SPLINE
SPL {X  -138.661, Y  +302.689, Z    +0.000, E1  +316.811, E3 -159767.577}
SPL {X  -154.202, Y  +339.857, Z    +0.000, E1  +330.366, E3 -159785.230}
SPL {X  -158.556, Y  +361.128, Z    +0.000, E1  +342.470, E3 -159789.751}
SPL {X  -159.866, Y  +376.206, Z    +0.000, E1  +353.031, E3 -159791.280}
SPL {X  -159.990, Y  +384.326, Z    +0.000, E1  +359.760, E3 -159791.553}
SPL {X  -159.990, Y  +385.649, Z    +0.000, E1  +361.559, E3 -159791.566}
SPL {X  -159.990, Y  +388.306, Z    +0.000, E1  +365.901, E3 -159791.637}
SPL {X  -159.990, Y  +392.624, Z    +0.000, E1  +373.655, E3 -159791.887}
SPL {X  -159.990, Y  +398.511, Z    +0.000, E1  +384.979, E3 -159792.467}
SPL {X  -159.990, Y  +405.629, Z    +0.000, E1  +396.596, E3 -159793.598}
SPL {X  -159.990, Y  +418.631, Z    +0.000, E1  +410.627, E3 -159796.545}
SPL {X  -159.990, Y  +468.459, Z    +0.000, E1  +425.348, E3 -159816.088}
SPL {X  -159.990, Y  +601.948, Z    +0.000, E1  +428.261, E3 -159902.214}
SPL {X  -159.990, Y  +614.867, Z    +0.000, E1  +428.239, E3 -159913.213}
SPL {X  -159.990, Y  +627.954, Z    +0.000, E1  +428.256, E3 -159924.257}
SPL {X  -159.990, Y  +640.176, Z    +0.000, E1  +428.239, E3 -159934.636}
SPL {X  -159.990, Y  +653.116, Z    +0.000, E1  +428.255, E3 -159945.568}
SPL {X  -159.990, Y  +665.424, Z    +0.000, E1  +428.236, E3 -159956.032}
SPL {X  -159.958, Y  +674.683, Z    +0.000, E1  +428.238, E3 -159963.881}
SPL {X  -159.269, Y  +686.675, Z    +0.000, E1  +428.163, E3 -159974.758}
SPL {X  -158.119, Y  +695.895, Z    +0.000, E1  +428.003, E3 -159983.799}
SPL {X  -156.550, Y  +704.498, Z    +0.000, E1  +427.821, E3 -159992.689}
SPL {X  -153.468, Y  +716.715, Z    +0.000, E1  +427.444, E3 -160006.152}
SPL {X  -149.840, Y  +727.578, Z    +0.000, E1  +426.935, E3 -160019.028}
SPL {X  -145.768, Y  +737.444, Z    +0.000, E1  +426.379, E3 -160031.330}
SPL {X  -141.751, Y  +745.686, Z    +0.000, E1  +425.756, E3 -160042.146}
SPL {X  -138.928, Y  +750.847, Z    +0.000, E1  +425.305, E3 -160049.116}
SPL {X  -136.328, Y  +755.234, Z    +0.000, E1  +424.898, E3 -160055.106}
SPL {X  -132.717, Y  +760.848, Z    +0.000, E1  +424.322, E3 -160062.879}
SPL {X  -128.512, Y  +766.796, Z    +0.000, E1  +423.597, E3 -160071.234}
SPL {X   -99.023, Y  +797.163, Z    +0.000, E1  +413.965, E3 -160173.063}
ENDSPLINE

SPLINE
SPL {X  -130.021, Y  +764.727, Z    +0.000, E1  +405.990, E3 -160312.582}
SPL {X  -148.409, Y  +731.264, Z    +0.000, E1  +396.685, E3 -160336.296}
SPL {X  -155.017, Y  +711.078, Z    +0.000, E1  +387.846, E3 -160343.357}
SPL {X  -158.217, Y  +695.254, Z    +0.000, E1  +378.896, E3 -160346.800}
SPL {X  -159.762, Y  +680.037, Z    +0.000, E1  +368.585, E3 -160348.517}
SPL {X  -159.990, Y  +669.745, Z    +0.000, E1  +360.389, E3 -160348.939}
SPL {X  -159.990, Y  +666.879, Z    +0.000, E1  +356.292, E3 -160348.990}
SPL {X  -159.990, Y  +662.620, Z    +0.000, E1  +348.758, E3 -160349.191}
SPL {X  -159.990, Y  +657.714, Z    +0.000, E1  +339.502, E3 -160349.612}
SPL {X  -159.990, Y  +651.038, Z    +0.000, E1  +327.797, E3 -160350.515}
SPL {X  -159.990, Y  +637.243, Z    +0.000, E1  +311.500, E3 -160353.640}
SPL {X  -159.990, Y  +579.875, Z    +0.000, E1  +294.421, E3 -160376.499}
SPL {X  -159.990, Y  +453.091, Z    +0.000, E1  +291.862, E3 -160459.468}
SPL {X  -159.990, Y  +439.299, Z    +0.000, E1  +291.885, E3 -160471.281}
SPL {X  -159.990, Y  +424.060, Z    +0.000, E1  +291.860, E3 -160484.229}
SPL {X  -159.990, Y  +408.047, Z    +0.000, E1  +291.885, E3 -160497.935}
SPL {X  -159.990, Y  +395.904, Z    +0.000, E1  +291.881, E3 -160508.271}
SPL {X  -157.896, Y  +356.699, Z    +0.000, E1  +289.725, E3 -160520.581}
SPL {X  -156.475, Y  +349.148, Z    +0.000, E1  +290.612, E3 -160534.045}
SPL {X  -155.960, Y  +346.816, Z    +0.000, E1  +291.495, E3 -160543.206}
SPL {X  -154.913, Y  +342.515, Z    +0.000, E1  +292.501, E3 -160555.220}
SPL {X  -152.032, Y  +332.668, Z    +0.000, E1  +292.988, E3 -160567.211}
SPL {X  -149.782, Y  +326.266, Z    +0.000, E1  +293.308, E3 -160574.951}
SPL {X  -147.566, Y  +320.686, Z    +0.000, E1  +293.613, E3 -160581.888}
SPL {X  -144.472, Y  +313.764, Z    +0.000, E1  +294.050, E3 -160590.757}
SPL {X  -140.755, Y  +306.442, Z    +0.000, E1  +294.606, E3 -160600.472}
SPL {X  -137.162, Y  +300.138, Z    +0.000, E1  +295.180, E3 -160609.080}
SPL {X  -132.996, Y  +293.568, Z    +0.000, E1  +295.842, E3 -160618.215}
SPL {X  -128.628, Y  +287.360, Z    +0.000, E1  +296.617, E3 -160627.016}
SPL {X   -99.903, Y  +257.535, Z    +0.000, E1  +308.539, E3 -160775.879}
ENDSPLINE

SPLINE
SPL {X  -141.433, Y  +307.709, Z    +0.000, E1  +318.157, E3 -160885.676}
SPL {X  -154.202, Y  +339.857, Z    +0.000, E1  +330.366, E3 -160899.515}
SPL {X  -158.556, Y  +361.128, Z    +0.000, E1  +342.470, E3 -160904.037}
SPL {X  -159.663, Y  +372.278, Z    +0.000, E1  +350.186, E3 -160905.319}
SPL {X  -159.986, Y  +381.388, Z    +0.000, E1  +357.201, E3 -160905.790}
SPL {X  -159.990, Y  +384.492, Z    +0.000, E1  +359.986, E3 -160905.840}
SPL {X  -159.990, Y  +385.649, Z    +0.000, E1  +361.559, E3 -160905.851}
SPL {X  -159.990, Y  +389.563, Z    +0.000, E1  +367.931, E3 -160905.984}
SPL {X  -159.990, Y  +396.421, Z    +0.000, E1  +380.831, E3 -160906.529}
SPL {X  -159.990, Y  +405.629, Z    +0.000, E1  +396.596, E3 -160907.883}
SPL {X  -159.990, Y  +418.631, Z    +0.000, E1  +410.627, E3 -160910.831}
SPL {X  -159.990, Y  +468.459, Z    +0.000, E1  +425.348, E3 -160930.374}
SPL {X  -159.990, Y  +601.948, Z    +0.000, E1  +428.261, E3 -161016.500}
SPL {X  -159.990, Y  +619.726, Z    +0.000, E1  +428.262, E3 -161031.561}
SPL {X  -159.990, Y  +636.530, Z    +0.000, E1  +428.257, E3 -161045.797}
SPL {X  -159.990, Y  +648.825, Z    +0.000, E1  +428.237, E3 -161056.256}
SPL {X  -159.990, Y  +661.441, Z    +0.000, E1  +428.256, E3 -161066.904}
SPL {X  -159.958, Y  +674.683, Z    +0.000, E1  +428.238, E3 -161078.166}
SPL {X  -159.269, Y  +686.675, Z    +0.000, E1  +428.163, E3 -161089.044}
SPL {X  -157.606, Y  +699.018, Z    +0.000, E1  +427.957, E3 -161101.228}
SPL {X  -155.210, Y  +710.317, Z    +0.000, E1  +427.656, E3 -161113.268}
SPL {X  -152.048, Y  +721.282, Z    +0.000, E1  +427.243, E3 -161125.760}
SPL {X  -148.485, Y  +731.073, Z    +0.000, E1  +426.748, E3 -161137.609}
SPL {X  -145.075, Y  +738.953, Z    +0.000, E1  +426.252, E3 -161147.601}
SPL {X  -141.751, Y  +745.686, Z    +0.000, E1  +425.756, E3 -161156.432}
SPL {X  -138.928, Y  +750.847, Z    +0.000, E1  +425.305, E3 -161163.401}
SPL {X  -136.328, Y  +755.234, Z    +0.000, E1  +424.898, E3 -161169.392}
SPL {X  -132.717, Y  +760.848, Z    +0.000, E1  +424.322, E3 -161177.165}
SPL {X  -128.512, Y  +766.796, Z    +0.000, E1  +423.597, E3 -161185.519}
SPL {X   -99.023, Y  +797.163, Z    +0.000, E1  +413.965, E3 -161287.349}
ENDSPLINE

SPLINE
SPL {X  -130.021, Y  +764.727, Z    +0.000, E1  +405.990, E3 -161426.868}
SPL {X  -148.409, Y  +731.264, Z    +0.000, E1  +396.685, E3 -161450.582}
SPL {X  -155.017, Y  +711.078, Z    +0.000, E1  +387.846, E3 -161457.643}
SPL {X  -158.217, Y  +695.254, Z    +0.000, E1  +378.896, E3 -161461.086}
SPL {X  -159.762, Y  +680.037, Z    +0.000, E1  +368.585, E3 -161462.802}
SPL {X  -159.990, Y  +671.255, Z    +0.000, E1  +361.602, E3 -161463.208}
SPL {X  -159.990, Y  +669.426, Z    +0.000, E1  +359.932, E3 -161463.228}
SPL {X  -159.990, Y  +666.879, Z    +0.000, E1  +356.292, E3 -161463.276}
SPL {X  -159.990, Y  +662.620, Z    +0.000, E1  +348.758, E3 -161463.477}
SPL {X  -159.990, Y  +657.714, Z    +0.000, E1  +339.502, E3 -161463.898}
SPL {X  -159.990, Y  +651.038, Z    +0.000, E1  +327.797, E3 -161464.800}
SPL {X  -159.990, Y  +637.243, Z    +0.000, E1  +311.500, E3 -161467.926}
SPL {X  -159.990, Y  +579.875, Z    +0.000, E1  +294.421, E3 -161490.784}
SPL {X  -159.990, Y  +458.824, Z    +0.000, E1  +291.885, E3 -161568.920}
SPL {X  -159.990, Y  +443.948, Z    +0.000, E1  +291.858, E3 -161581.543}
SPL {X  -159.990, Y  +424.060, Z    +0.000, E1  +291.860, E3 -161598.515}
SPL {X  -159.990, Y  +408.047, Z    +0.000, E1  +291.885, E3 -161612.221}
SPL {X  -159.990, Y  +395.904, Z    +0.000, E1  +291.881, E3 -161622.557}
SPL {X  -157.896, Y  +356.699, Z    +0.000, E1  +289.725, E3 -161634.866}
SPL {X  -156.475, Y  +349.148, Z    +0.000, E1  +290.612, E3 -161648.330}
SPL {X  -155.786, Y  +346.063, Z    +0.000, E1  +291.892, E3 -161661.625}
SPL {X  -154.401, Y  +340.583, Z    +0.000, E1  +292.675, E3 -161672.322}
SPL {X  -152.032, Y  +332.668, Z    +0.000, E1  +292.988, E3 -161681.497}
SPL {X  -148.460, Y  +322.864, Z    +0.000, E1  +293.452, E3 -161693.380}
SPL {X  -144.472, Y  +313.764, Z    +0.000, E1  +294.050, E3 -161705.043}
SPL {X  -140.755, Y  +306.442, Z    +0.000, E1  +294.606, E3 -161714.758}
SPL {X  -137.162, Y  +300.138, Z    +0.000, E1  +295.180, E3 -161723.366}
SPL {X  -132.996, Y  +293.568, Z    +0.000, E1  +295.842, E3 -161732.500}
SPL {X  -128.628, Y  +287.360, Z    +0.000, E1  +296.617, E3 -161741.301}
SPL {X   -98.696, Y  +256.580, Z    +0.000, E1  +308.006, E3 -161878.420}
ENDSPLINE

SPLINE
SPL {X  -138.661, Y  +302.689, Z    +0.000, E1  +316.811, E3 -161996.148}
SPL {X  -154.202, Y  +339.857, Z    +0.000, E1  +330.366, E3 -162013.801}
SPL {X  -158.556, Y  +361.128, Z    +0.000, E1  +342.470, E3 -162018.323}
SPL {X  -159.866, Y  +376.206, Z    +0.000, E1  +353.031, E3 -162019.852}
SPL {X  -159.990, Y  +384.789, Z    +0.000, E1  +360.146, E3 -162020.129}
SPL {X  -159.990, Y  +389.563, Z    +0.000, E1  +367.931, E3 -162020.269}
SPL {X  -159.990, Y  +396.421, Z    +0.000, E1  +380.831, E3 -162020.814}
SPL {X  -159.990, Y  +405.629, Z    +0.000, E1  +396.596, E3 -162022.169}
SPL {X  -159.990, Y  +417.919, Z    +0.000, E1  +410.108, E3 -162024.895}
SPL {X  -159.990, Y  +464.219, Z    +0.000, E1  +424.792, E3 -162042.954}
SPL {X  -159.990, Y  +601.948, Z    +0.000, E1  +428.261, E3 -162130.786}
SPL {X  -159.990, Y  +614.867, Z    +0.000, E1  +428.239, E3 -162141.784}
SPL {X  -159.990, Y  +627.954, Z    +0.000, E1  +428.256, E3 -162152.829}
SPL {X  -159.990, Y  +640.176, Z    +0.000, E1  +428.239, E3 -162163.207}
SPL {X  -159.990, Y  +653.116, Z    +0.000, E1  +428.255, E3 -162174.139}
SPL {X  -159.990, Y  +665.424, Z    +0.000, E1  +428.236, E3 -162184.603}
SPL {X  -159.958, Y  +674.683, Z    +0.000, E1  +428.238, E3 -162192.452}
SPL {X  -159.269, Y  +686.675, Z    +0.000, E1  +428.163, E3 -162203.330}
SPL {X  -157.606, Y  +699.018, Z    +0.000, E1  +427.957, E3 -162215.513}
SPL {X  -155.210, Y  +710.317, Z    +0.000, E1  +427.656, E3 -162227.553}
SPL {X  -152.048, Y  +721.282, Z    +0.000, E1  +427.243, E3 -162240.046}
SPL {X  -148.485, Y  +731.073, Z    +0.000, E1  +426.748, E3 -162251.895}
SPL {X  -145.075, Y  +738.953, Z    +0.000, E1  +426.252, E3 -162261.887}
SPL {X  -141.751, Y  +745.686, Z    +0.000, E1  +425.756, E3 -162270.718}
SPL {X  -138.928, Y  +750.847, Z    +0.000, E1  +425.305, E3 -162277.687}
SPL {X  -136.328, Y  +755.234, Z    +0.000, E1  +424.898, E3 -162283.677}
SPL {X  -132.717, Y  +760.848, Z    +0.000, E1  +424.322, E3 -162291.450}
SPL {X  -128.512, Y  +766.796, Z    +0.000, E1  +423.597, E3 -162299.805}
SPL {X   -99.023, Y  +797.163, Z    +0.000, E1  +413.965, E3 -162401.635}
ENDSPLINE

SPLINE
SPL {X  -130.021, Y  +764.727, Z    +0.000, E1  +405.990, E3 -162541.154}
SPL {X  -148.409, Y  +731.264, Z    +0.000, E1  +396.685, E3 -162564.867}
SPL {X  -155.017, Y  +711.078, Z    +0.000, E1  +387.846, E3 -162571.928}
SPL {X  -158.217, Y  +695.254, Z    +0.000, E1  +378.896, E3 -162575.371}
SPL {X  -159.762, Y  +680.037, Z    +0.000, E1  +368.585, E3 -162577.088}
SPL {X  -159.990, Y  +671.255, Z    +0.000, E1  +361.602, E3 -162577.494}
SPL {X  -159.990, Y  +669.148, Z    +0.000, E1  +359.679, E3 -162577.516}
SPL {X  -159.990, Y  +666.130, Z    +0.000, E1  +354.946, E3 -162577.582}
SPL {X  -159.990, Y  +662.620, Z    +0.000, E1  +348.758, E3 -162577.762}
SPL {X  -159.990, Y  +657.714, Z    +0.000, E1  +339.502, E3 -162578.184}
SPL {X  -159.990, Y  +651.038, Z    +0.000, E1  +327.797, E3 -162579.086}
SPL {X  -159.990, Y  +637.243, Z    +0.000, E1  +311.500, E3 -162582.211}
SPL {X  -159.990, Y  +579.875, Z    +0.000, E1  +294.421, E3 -162605.070}
SPL {X  -159.990, Y  +453.091, Z    +0.000, E1  +291.862, E3 -162688.039}
SPL {X  -159.990, Y  +439.299, Z    +0.000, E1  +291.885, E3 -162699.852}
SPL {X  -159.990, Y  +424.060, Z    +0.000, E1  +291.860, E3 -162712.800}
SPL {X  -159.990, Y  +408.047, Z    +0.000, E1  +291.885, E3 -162726.507}
SPL {X  -159.990, Y  +395.904, Z    +0.000, E1  +291.881, E3 -162736.843}
SPL {X  -157.896, Y  +356.699, Z    +0.000, E1  +289.725, E3 -162749.152}
SPL {X  -156.475, Y  +349.148, Z    +0.000, E1  +290.612, E3 -162762.616}
SPL {X  -155.786, Y  +346.063, Z    +0.000, E1  +291.892, E3 -162775.911}
SPL {X  -154.401, Y  +340.583, Z    +0.000, E1  +292.675, E3 -162786.607}
SPL {X  -152.032, Y  +332.668, Z    +0.000, E1  +292.988, E3 -162795.783}
SPL {X  -149.782, Y  +326.266, Z    +0.000, E1  +293.308, E3 -162803.523}
SPL {X  -146.798, Y  +318.884, Z    +0.000, E1  +293.699, E3 -162812.703}
SPL {X  -143.755, Y  +312.276, Z    +0.000, E1  +294.175, E3 -162821.313}
SPL {X  -140.755, Y  +306.442, Z    +0.000, E1  +294.606, E3 -162829.044}
SPL {X  -137.162, Y  +300.138, Z    +0.000, E1  +295.180, E3 -162837.652}
SPL {X  -134.303, Y  +295.555, Z    +0.000, E1  +295.659, E3 -162844.033}
SPL {X  -132.067, Y  +292.194, Z    +0.000, E1  +296.034, E3 -162848.764}
SPL {X  -128.628, Y  +287.360, Z    +0.000, E1  +296.617, E3 -162855.587}
SPL {X   -99.903, Y  +257.535, Z    +0.000, E1  +308.539, E3 -163004.450}
ENDSPLINE

SPLINE
SPL {X  -141.433, Y  +307.709, Z    +0.000, E1  +318.157, E3 -163114.247}
SPL {X  -151.246, Y  +330.333, Z    +0.000, E1  +326.099, E3 -163125.138}
SPL {X  -155.793, Y  +346.095, Z    +0.000, E1  +333.603, E3 -163129.796}
SPL {X  -158.556, Y  +361.128, Z    +0.000, E1  +342.470, E3 -163132.609}
SPL {X  -159.866, Y  +376.206, Z    +0.000, E1  +353.031, E3 -163134.138}
SPL {X  -159.990, Y  +384.326, Z    +0.000, E1  +359.760, E3 -163134.410}
SPL {X  -159.990, Y  +385.649, Z    +0.000, E1  +361.559, E3 -163134.423}
SPL {X  -159.990, Y  +388.306, Z    +0.000, E1  +365.901, E3 -163134.494}
SPL {X  -159.990, Y  +392.624, Z    +0.000, E1  +373.655, E3 -163134.744}
SPL {X  -159.990, Y  +398.511, Z    +0.000, E1  +384.979, E3 -163135.324}
SPL {X  -159.990, Y  +405.629, Z    +0.000, E1  +396.596, E3 -163136.455}
SPL {X  -159.990, Y  +418.631, Z    +0.000, E1  +410.627, E3 -163139.402}
SPL {X  -159.990, Y  +468.459, Z    +0.000, E1  +425.348, E3 -163158.945}
SPL {X  -159.990, Y  +601.948, Z    +0.000, E1  +428.261, E3 -163245.071}
SPL {X  -159.990, Y  +619.726, Z    +0.000, E1  +428.262, E3 -163260.132}
SPL {X  -159.990, Y  +636.530, Z    +0.000, E1  +428.257, E3 -163274.368}
SPL {X  -159.990, Y  +648.825, Z    +0.000, E1  +428.237, E3 -163284.827}
SPL {X  -159.990, Y  +661.441, Z    +0.000, E1  +428.256, E3 -163295.475}
SPL {X  -159.958, Y  +674.683, Z    +0.000, E1  +428.238, E3 -163306.738}
SPL {X  -159.269, Y  +686.675, Z    +0.000, E1  +428.163, E3 -163317.615}
SPL {X  -157.606, Y  +699.018, Z    +0.000, E1  +427.957, E3 -163329.799}
SPL {X  -155.210, Y  +710.317, Z    +0.000, E1  +427.656, E3 -163341.839}
SPL {X  -152.048, Y  +721.282, Z    +0.000, E1  +427.243, E3 -163354.332}
SPL {X  -148.485, Y  +731.073, Z    +0.000, E1  +426.748, E3 -163366.181}
SPL {X  -145.075, Y  +738.953, Z    +0.000, E1  +426.252, E3 -163376.172}
SPL {X  -141.751, Y  +745.686, Z    +0.000, E1  +425.756, E3 -163385.003}
SPL {X  -138.928, Y  +750.847, Z    +0.000, E1  +425.305, E3 -163391.973}
SPL {X  -136.328, Y  +755.234, Z    +0.000, E1  +424.898, E3 -163397.963}
SPL {X  -132.717, Y  +760.848, Z    +0.000, E1  +424.322, E3 -163405.736}
SPL {X  -128.512, Y  +766.796, Z    +0.000, E1  +423.597, E3 -163414.091}
SPL {X   -99.023, Y  +797.163, Z    +0.000, E1  +413.965, E3 -163515.920}
ENDSPLINE

SPLINE
SPL {X  -130.021, Y  +764.727, Z    +0.000, E1  +405.990, E3 -163655.440}
SPL {X  -148.409, Y  +731.264, Z    +0.000, E1  +396.685, E3 -163679.153}
SPL {X  -155.017, Y  +711.078, Z    +0.000, E1  +387.846, E3 -163686.214}
SPL {X  -158.217, Y  +695.254, Z    +0.000, E1  +378.896, E3 -163689.657}
SPL {X  -159.762, Y  +680.037, Z    +0.000, E1  +368.585, E3 -163691.374}
SPL {X  -159.990, Y  +671.255, Z    +0.000, E1  +361.602, E3 -163691.779}
SPL {X  -159.990, Y  +669.426, Z    +0.000, E1  +359.932, E3 -163691.799}
SPL {X  -159.990, Y  +666.879, Z    +0.000, E1  +356.292, E3 -163691.847}
SPL {X  -159.990, Y  +662.620, Z    +0.000, E1  +348.758, E3 -163692.048}
SPL {X  -159.990, Y  +657.714, Z    +0.000, E1  +339.502, E3 -163692.469}
SPL {X  -159.990, Y  +651.038, Z    +0.000, E1  +327.797, E3 -163693.372}
SPL {X  -159.990, Y  +637.243, Z    +0.000, E1  +311.500, E3 -163696.497}
SPL {X  -159.990, Y  +579.875, Z    +0.000, E1  +294.421, E3 -163719.356}
SPL {X  -159.990, Y  +453.091, Z    +0.000, E1  +291.862, E3 -163802.325}
SPL {X  -159.990, Y  +434.933, Z    +0.000, E1  +291.864, E3 -163817.819}
SPL {X  -159.990, Y  +420.071, Z    +0.000, E1  +291.886, E3 -163830.545}
SPL {X  -159.990, Y  +408.047, Z    +0.000, E1  +291.885, E3 -163840.792}
SPL {X  -159.990, Y  +395.904, Z    +0.000, E1  +291.881, E3 -163851.128}
SPL {X  -157.896, Y  +356.699, Z    +0.000, E1  +289.725, E3 -163863.438}
SPL {X  -156.475, Y  +349.148, Z    +0.000, E1  +290.612, E3 -163876.902}
SPL {X  -155.786, Y  +346.063, Z    +0.000, E1  +291.892, E3 -163890.196}
SPL {X  -153.671, Y  +337.981, Z    +0.000, E1  +292.746, E3 -163903.816}
SPL {X  -150.407, Y  +327.960, Z    +0.000, E1  +293.203, E3 -163915.705}
SPL {X  -146.798, Y  +318.884, Z    +0.000, E1  +293.699, E3 -163926.989}
SPL {X  -142.741, Y  +310.238, Z    +0.000, E1  +294.301, E3 -163938.248}
SPL {X  -139.838, Y  +304.768, Z    +0.000, E1  +294.773, E3 -163945.631}
SPL {X  -137.162, Y  +300.138, Z    +0.000, E1  +295.180, E3 -163951.937}
SPL {X  -132.996, Y  +293.568, Z    +0.000, E1  +295.842, E3 -163961.072}
SPL {X  -128.628, Y  +287.360, Z    +0.000, E1  +296.617, E3 -163969.873}
SPL {X   -98.696, Y  +256.580, Z    +0.000, E1  +308.006, E3 -164106.991}
ENDSPLINE

SPLINE
SPL {X  -138.661, Y  +302.689, Z    +0.000, E1  +316.811, E3 -164224.720}
SPL {X  -154.202, Y  +339.857, Z    +0.000, E1  +330.366, E3 -164242.373}
SPL {X  -158.556, Y  +361.128, Z    +0.000, E1  +342.470, E3 -164246.894}
SPL {X  -159.663, Y  +372.278, Z    +0.000, E1  +350.186, E3 -164248.176}
SPL {X  -159.986, Y  +381.388, Z    +0.000, E1  +357.201, E3 -164248.647}
SPL {X  -159.990, Y  +384.492, Z    +0.000, E1  +359.986, E3 -164248.697}
SPL {X  -159.990, Y  +385.649, Z    +0.000, E1  +361.559, E3 -164248.709}
SPL {X  -159.990, Y  +389.563, Z    +0.000, E1  +367.931, E3 -164248.841}
SPL {X  -159.990, Y  +396.421, Z    +0.000, E1  +380.831, E3 -164249.386}
SPL {X  -159.990, Y  +405.629, Z    +0.000, E1  +396.596, E3 -164250.740}
SPL {X  -159.990, Y  +418.631, Z    +0.000, E1  +410.627, E3 -164253.688}
SPL {X  -159.990, Y  +468.459, Z    +0.000, E1  +425.348, E3 -164273.231}
SPL {X  -159.990, Y  +601.948, Z    +0.000, E1  +428.261, E3 -164359.357}
SPL {X  -159.990, Y  +619.726, Z    +0.000, E1  +428.262, E3 -164374.418}
SPL {X  -159.990, Y  +636.530, Z    +0.000, E1  +428.257, E3 -164388.654}
SPL {X  -159.990, Y  +648.825, Z    +0.000, E1  +428.237, E3 -164399.113}
SPL {X  -159.990, Y  +661.441, Z    +0.000, E1  +428.256, E3 -164409.761}
SPL {X  -159.958, Y  +674.683, Z    +0.000, E1  +428.238, E3 -164421.024}
SPL {X  -159.269, Y  +686.675, Z    +0.000, E1  +428.163, E3 -164431.901}
SPL {X  -158.119, Y  +695.895, Z    +0.000, E1  +428.003, E3 -164440.942}
SPL {X  -156.550, Y  +704.498, Z    +0.000, E1  +427.821, E3 -164449.832}
SPL {X  -154.561, Y  +712.826, Z    +0.000, E1  +427.549, E3 -164458.963}
SPL {X  -152.048, Y  +721.282, Z    +0.000, E1  +427.243, E3 -164468.617}
SPL {X  -148.485, Y  +731.073, Z    +0.000, E1  +426.748, E3 -164480.466}
SPL {X  -145.075, Y  +738.953, Z    +0.000, E1  +426.252, E3 -164490.458}
SPL {X  -141.751, Y  +745.686, Z    +0.000, E1  +425.756, E3 -164499.289}
SPL {X  -138.928, Y  +750.847, Z    +0.000, E1  +425.305, E3 -164506.258}
SPL {X  -136.328, Y  +755.234, Z    +0.000, E1  +424.898, E3 -164512.249}
SPL {X  -132.717, Y  +760.848, Z    +0.000, E1  +424.322, E3 -164520.022}
SPL {X  -128.512, Y  +766.796, Z    +0.000, E1  +423.597, E3 -164528.376}
SPL {X   -99.023, Y  +797.163, Z    +0.000, E1  +413.965, E3 -164630.206}
ENDSPLINE

SPLINE
SPL {X  -130.021, Y  +764.727, Z    +0.000, E1  +405.990, E3 -164769.725}
SPL {X  -148.409, Y  +731.264, Z    +0.000, E1  +396.685, E3 -164793.439}
SPL {X  -155.017, Y  +711.078, Z    +0.000, E1  +387.846, E3 -164800.500}
SPL {X  -158.217, Y  +695.254, Z    +0.000, E1  +378.896, E3 -164803.943}
SPL {X  -159.762, Y  +680.037, Z    +0.000, E1  +368.585, E3 -164805.660}
SPL {X  -159.990, Y  +671.255, Z    +0.000, E1  +361.602, E3 -164806.065}
SPL {X  -159.990, Y  +669.148, Z    +0.000, E1  +359.679, E3 -164806.088}
SPL {X  -159.990, Y  +666.130, Z    +0.000, E1  +354.946, E3 -164806.154}
SPL {X  -159.990, Y  +662.620, Z    +0.000, E1  +348.758, E3 -164806.334}
SPL {X  -159.990, Y  +657.714, Z    +0.000, E1  +339.502, E3 -164806.755}
SPL {X  -159.990, Y  +651.038, Z    +0.000, E1  +327.797, E3 -164807.658}
SPL {X  -159.990, Y  +637.243, Z    +0.000, E1  +311.500, E3 -164810.783}
SPL {X  -159.990, Y  +579.875, Z    +0.000, E1  +294.421, E3 -164833.641}
SPL {X  -159.990, Y  +453.091, Z    +0.000, E1  +291.862, E3 -164916.611}
SPL {X  -159.990, Y  +439.299, Z    +0.000, E1  +291.885, E3 -164928.424}
SPL {X  -159.990, Y  +424.060, Z    +0.000, E1  +291.860, E3 -164941.372}
SPL {X  -159.990, Y  +408.047, Z    +0.000, E1  +291.885, E3 -164955.078}
SPL {X  -159.990, Y  +395.904, Z    +0.000, E1  +291.881, E3 -164965.414}
SPL {X  -157.896, Y  +356.699, Z    +0.000, E1  +289.725, E3 -164977.724}
SPL {X  -156.475, Y  +349.148, Z    +0.000, E1  +290.612, E3 -164991.188}
SPL {X  -155.786, Y  +346.063, Z    +0.000, E1  +291.892, E3 -165004.482}
SPL {X  -154.401, Y  +340.583, Z    +0.000, E1  +292.675, E3 -165015.179}
SPL {X  -152.032, Y  +332.668, Z    +0.000, E1  +292.988, E3 -165024.354}
SPL {X  -149.782, Y  +326.266, Z    +0.000, E1  +293.308, E3 -165032.094}
SPL {X  -146.798, Y  +318.884, Z    +0.000, E1  +293.699, E3 -165041.275}
SPL {X  -143.755, Y  +312.276, Z    +0.000, E1  +294.175, E3 -165049.884}
SPL {X  -140.755, Y  +306.442, Z    +0.000, E1  +294.606, E3 -165057.615}
SPL {X  -137.162, Y  +300.138, Z    +0.000, E1  +295.180, E3 -165066.223}
SPL {X  -134.303, Y  +295.555, Z    +0.000, E1  +295.659, E3 -165072.604}
SPL {X  -132.067, Y  +292.194, Z    +0.000, E1  +296.034, E3 -165077.336}
SPL {X  -128.628, Y  +287.360, Z    +0.000, E1  +296.617, E3 -165084.159}
SPL {X   -98.696, Y  +256.580, Z    +0.000, E1  +308.006, E3 -165221.277}
ENDSPLINE

SPLINE
SPL {X  -138.661, Y  +302.689, Z    +0.000, E1  +316.811, E3 -165339.005}
SPL {X  -154.202, Y  +339.857, Z    +0.000, E1  +330.366, E3 -165356.658}
SPL {X  -158.556, Y  +361.128, Z    +0.000, E1  +342.470, E3 -165361.180}
SPL {X  -159.866, Y  +376.206, Z    +0.000, E1  +353.031, E3 -165362.709}
SPL {X  -159.990, Y  +384.326, Z    +0.000, E1  +359.760, E3 -165362.982}
SPL {X  -159.990, Y  +385.649, Z    +0.000, E1  +361.559, E3 -165362.994}
SPL {X  -159.990, Y  +389.563, Z    +0.000, E1  +367.931, E3 -165363.127}
SPL {X  -159.990, Y  +396.421, Z    +0.000, E1  +380.831, E3 -165363.672}
SPL {X  -159.990, Y  +405.629, Z    +0.000, E1  +396.596, E3 -165365.026}
SPL {X  -159.990, Y  +418.631, Z    +0.000, E1  +410.627, E3 -165367.973}
SPL {X  -159.990, Y  +468.459, Z    +0.000, E1  +425.348, E3 -165387.517}
SPL {X  -159.990, Y  +601.948, Z    +0.000, E1  +428.261, E3 -165473.643}
SPL {X  -159.990, Y  +619.726, Z    +0.000, E1  +428.262, E3 -165488.704}
SPL {X  -159.990, Y  +636.530, Z    +0.000, E1  +428.257, E3 -165502.940}
SPL {X  -159.990, Y  +653.116, Z    +0.000, E1  +428.255, E3 -165516.996}
SPL {X  -159.990, Y  +665.424, Z    +0.000, E1  +428.236, E3 -165527.461}
SPL {X  -159.958, Y  +674.683, Z    +0.000, E1  +428.238, E3 -165535.309}
SPL {X  -159.269, Y  +686.675, Z    +0.000, E1  +428.163, E3 -165546.187}
SPL {X  -158.119, Y  +695.895, Z    +0.000, E1  +428.003, E3 -165555.227}
SPL {X  -156.550, Y  +704.498, Z    +0.000, E1  +427.821, E3 -165564.118}
SPL {X  -154.561, Y  +712.826, Z    +0.000, E1  +427.549, E3 -165573.248}
SPL {X  -152.048, Y  +721.282, Z    +0.000, E1  +427.243, E3 -165582.903}
SPL {X  -148.485, Y  +731.073, Z    +0.000, E1  +426.748, E3 -165594.752}
SPL {X  -145.075, Y  +738.953, Z    +0.000, E1  +426.252, E3 -165604.744}
SPL {X  -141.751, Y  +745.686, Z    +0.000, E1  +425.756, E3 -165613.575}
SPL {X  -138.928, Y  +750.847, Z    +0.000, E1  +425.305, E3 -165620.544}
SPL {X  -135.390, Y  +756.743, Z    +0.000, E1  +424.775, E3 -165628.576}
SPL {X  -132.002, Y  +761.900, Z    +0.000, E1  +424.179, E3 -165635.808}
SPL {X  -128.512, Y  +766.796, Z    +0.000, E1  +423.597, E3 -165642.662}
SPL {X   -99.023, Y  +797.163, Z    +0.000, E1  +413.965, E3 -165744.492}
ENDSPLINE

SPLINE
SPL {X  -130.021, Y  +764.727, Z    +0.000, E1  +405.990, E3 -165884.011}
SPL {X  -148.409, Y  +731.264, Z    +0.000, E1  +396.685, E3 -165907.725}
SPL {X  -155.017, Y  +711.078, Z    +0.000, E1  +387.846, E3 -165914.786}
SPL {X  -158.217, Y  +695.254, Z    +0.000, E1  +378.896, E3 -165918.228}
SPL {X  -159.524, Y  +683.703, Z    +0.000, E1  +371.166, E3 -165919.670}
SPL {X  -159.986, Y  +672.621, Z    +0.000, E1  +362.847, E3 -165920.312}
SPL {X  -159.990, Y  +669.148, Z    +0.000, E1  +359.679, E3 -165920.373}
SPL {X  -159.990, Y  +666.130, Z    +0.000, E1  +354.946, E3 -165920.439}
SPL {X  -159.990, Y  +662.620, Z    +0.000, E1  +348.758, E3 -165920.620}
SPL {X  -159.990, Y  +657.714, Z    +0.000, E1  +339.502, E3 -165921.041}
SPL {X  -159.990, Y  +651.038, Z    +0.000, E1  +327.797, E3 -165921.943}
SPL {X  -159.990, Y  +642.324, Z    +0.000, E1  +316.129, E3 -165923.678}
SPL {X  -159.990, Y  +634.003, Z    +0.000, E1  +308.893, E3 -165925.953}
SPL {X  -159.990, Y  +579.875, Z    +0.000, E1  +294.421, E3 -165947.927}
SPL {X  -159.990, Y  +453.091, Z    +0.000, E1  +291.862, E3 -166030.897}
SPL {X  -159.990, Y  +434.933, Z    +0.000, E1  +291.864, E3 -166046.390}
SPL {X  -159.990, Y  +420.071, Z    +0.000, E1  +291.886, E3 -166059.116}
SPL {X  -159.990, Y  +408.047, Z    +0.000, E1  +291.885, E3 -166069.364}
SPL {X  -159.990, Y  +395.904, Z    +0.000, E1  +291.881, E3 -166079.700}
SPL {X  -157.896, Y  +356.699, Z    +0.000, E1  +289.725, E3 -166092.009}
SPL {X  -156.475, Y  +349.148, Z    +0.000, E1  +290.612, E3 -166105.473}
SPL {X  -155.786, Y  +346.063, Z    +0.000, E1  +291.892, E3 -166118.768}
SPL {X  -154.401, Y  +340.583, Z    +0.000, E1  +292.675, E3 -166129.464}
SPL {X  -152.032, Y  +332.668, Z    +0.000, E1  +292.988, E3 -166138.640}
SPL {X  -148.460, Y  +322.864, Z    +0.000, E1  +293.452, E3 -166150.523}
SPL {X  -144.472, Y  +313.764, Z    +0.000, E1  +294.050, E3 -166162.186}
SPL {X  -140.755, Y  +306.442, Z    +0.000, E1  +294.606, E3 -166171.901}
SPL {X  -137.162, Y  +300.138, Z    +0.000, E1  +295.180, E3 -166180.509}
SPL {X  -134.303, Y  +295.555, Z    +0.000, E1  +295.659, E3 -166186.890}
SPL {X  -131.069, Y  +290.753, Z    +0.000, E1  +296.178, E3 -166193.623}
SPL {X  -127.815, Y  +286.271, Z    +0.000, E1  +296.784, E3 -166200.012}
SPL {X   -99.903, Y  +257.535, Z    +0.000, E1  +308.539, E3 -166347.307}
ENDSPLINE

SPLINE
SPL {X  -141.433, Y  +307.709, Z    +0.000, E1  +318.157, E3 -166457.104}
SPL {X  -154.202, Y  +339.857, Z    +0.000, E1  +330.366, E3 -166470.944}
SPL {X  -158.556, Y  +361.128, Z    +0.000, E1  +342.470, E3 -166475.466}
SPL {X  -159.663, Y  +372.278, Z    +0.000, E1  +350.186, E3 -166476.747}
SPL {X  -159.986, Y  +381.388, Z    +0.000, E1  +357.201, E3 -166477.218}
SPL {X  -159.990, Y  +384.492, Z    +0.000, E1  +359.986, E3 -166477.269}
SPL {X  -159.990, Y  +385.649, Z    +0.000, E1  +361.559, E3 -166477.280}
SPL {X  -159.990, Y  +389.563, Z    +0.000, E1  +367.931, E3 -166477.412}
SPL {X  -159.990, Y  +396.421, Z    +0.000, E1  +380.831, E3 -166477.957}
SPL {X  -159.990, Y  +405.629, Z    +0.000, E1  +396.596, E3 -166479.312}
SPL {X  -159.990, Y  +418.631, Z    +0.000, E1  +410.627, E3 -166482.259}
SPL {X  -159.990, Y  +468.459, Z    +0.000, E1  +425.348, E3 -166501.803}
SPL {X  -159.990, Y  +601.948, Z    +0.000, E1  +428.261, E3 -166587.929}
SPL {X  -159.990, Y  +619.726, Z    +0.000, E1  +428.262, E3 -166602.989}
SPL {X  -159.990, Y  +636.530, Z    +0.000, E1  +428.257, E3 -166617.225}
SPL {X  -159.990, Y  +648.825, Z    +0.000, E1  +428.237, E3 -166627.684}
SPL {X  -159.990, Y  +661.441, Z    +0.000, E1  +428.256, E3 -166638.332}
SPL {X  -159.958, Y  +674.683, Z    +0.000, E1  +428.238, E3 -166649.595}
SPL {X  -159.269, Y  +686.675, Z    +0.000, E1  +428.163, E3 -166660.472}
SPL {X  -158.119, Y  +695.895, Z    +0.000, E1  +428.003, E3 -166669.513}
SPL {X  -156.550, Y  +704.498, Z    +0.000, E1  +427.821, E3 -166678.403}
SPL {X  -154.561, Y  +712.826, Z    +0.000, E1  +427.549, E3 -166687.534}
SPL {X  -152.683, Y  +719.299, Z    +0.000, E1  +427.307, E3 -166694.908}
SPL {X  -149.840, Y  +727.578, Z    +0.000, E1  +426.935, E3 -166704.742}
SPL {X  -145.768, Y  +737.444, Z    +0.000, E1  +426.379, E3 -166717.044}
SPL {X  -141.751, Y  +745.686, Z    +0.000, E1  +425.756, E3 -166727.860}
SPL {X  -138.928, Y  +750.847, Z    +0.000, E1  +425.305, E3 -166734.830}
SPL {X  -136.328, Y  +755.234, Z    +0.000, E1  +424.898, E3 -166740.820}
SPL {X  -132.717, Y  +760.848, Z    +0.000, E1  +424.322, E3 -166748.593}
SPL {X  -128.512, Y  +766.796, Z    +0.000, E1  +423.597, E3 -166756.948}
SPL {X   -99.023, Y  +797.163, Z    +0.000, E1  +413.965, E3 -166858.777}
ENDSPLINE

SPLINE
SPL {X  -130.021, Y  +764.727, Z    +0.000, E1  +405.990, E3 -166998.297}
SPL {X  -148.409, Y  +731.264, Z    +0.000, E1  +396.685, E3 -167022.010}
SPL {X  -155.017, Y  +711.078, Z    +0.000, E1  +387.846, E3 -167029.071}
SPL {X  -158.217, Y  +695.254, Z    +0.000, E1  +378.896, E3 -167032.514}
SPL {X  -159.524, Y  +683.703, Z    +0.000, E1  +371.166, E3 -167033.956}
SPL {X  -159.986, Y  +672.621, Z    +0.000, E1  +362.847, E3 -167034.598}
SPL {X  -159.990, Y  +669.426, Z    +0.000, E1  +359.932, E3 -167034.656}
SPL {X  -159.990, Y  +666.879, Z    +0.000, E1  +356.292, E3 -167034.704}
SPL {X  -159.990, Y  +662.620, Z    +0.000, E1  +348.758, E3 -167034.905}
SPL {X  -159.990, Y  +657.714, Z    +0.000, E1  +339.502, E3 -167035.327}
SPL {X  -159.990, Y  +651.038, Z    +0.000, E1  +327.797, E3 -167036.229}
SPL {X  -159.990, Y  +637.243, Z    +0.000, E1  +311.500, E3 -167039.354}
SPL {X  -159.990, Y  +579.875, Z    +0.000, E1  +294.421, E3 -167062.213}
SPL {X  -159.990, Y  +453.091, Z    +0.000, E1  +291.862, E3 -167145.182}
SPL {X  -159.990, Y  +434.933, Z    +0.000, E1  +291.864, E3 -167160.676}
SPL {X  -159.990, Y  +420.071, Z    +0.000, E1  +291.886, E3 -167173.402}
SPL {X  -159.990, Y  +408.047, Z    +0.000, E1  +291.885, E3 -167183.650}
SPL {X  -159.990, Y  +395.904, Z    +0.000, E1  +291.881, E3 -167193.986}
SPL {X  -157.896, Y  +356.699, Z    +0.000, E1  +289.725, E3 -167206.295}
SPL {X  -156.475, Y  +349.148, Z    +0.000, E1  +290.612, E3 -167219.759}
SPL {X  -155.960, Y  +346.816, Z    +0.000, E1  +291.495, E3 -167228.920}
SPL {X  -154.913, Y  +342.515, Z    +0.000, E1  +292.501, E3 -167240.934}
SPL {X  -152.032, Y  +332.668, Z    +0.000, E1  +292.988, E3 -167252.926}
SPL {X  -148.460, Y  +322.864, Z    +0.000, E1  +293.452, E3 -167264.808}
SPL {X  -144.472, Y  +313.764, Z    +0.000, E1  +294.050, E3 -167276.472}
SPL {X  -140.755, Y  +306.442, Z    +0.000, E1  +294.606, E3 -167286.186}
SPL {X  -137.162, Y  +300.138, Z    +0.000, E1  +295.180, E3 -167294.795}
SPL {X  -134.303, Y  +295.555, Z    +0.000, E1  +295.659, E3 -167301.175}
SPL {X  -131.069, Y  +290.753, Z    +0.000, E1  +296.178, E3 -167307.909}
SPL {X  -127.815, Y  +286.271, Z    +0.000, E1  +296.784, E3 -167314.297}
SPL {X   -99.903, Y  +257.535, Z    +0.000, E1  +308.539, E3 -167461.593}
ENDSPLINE

SPLINE
SPL {X  -141.433, Y  +307.709, Z    +0.000, E1  +318.157, E3 -167571.390}
SPL {X  -154.202, Y  +339.857, Z    +0.000, E1  +330.366, E3 -167585.230}
SPL {X  -158.556, Y  +361.128, Z    +0.000, E1  +342.470, E3 -167589.751}
SPL {X  -159.663, Y  +372.278, Z    +0.000, E1  +350.186, E3 -167591.033}
SPL {X  -159.986, Y  +381.388, Z    +0.000, E1  +357.201, E3 -167591.504}
SPL {X  -159.990, Y  +384.492, Z    +0.000, E1  +359.986, E3 -167591.554}
SPL {X  -159.990, Y  +385.649, Z    +0.000, E1  +361.559, E3 -167591.566}
SPL {X  -159.990, Y  +389.563, Z    +0.000, E1  +367.931, E3 -167591.698}
SPL {X  -159.990, Y  +396.421, Z    +0.000, E1  +380.831, E3 -167592.243}
SPL {X  -159.990, Y  +405.629, Z    +0.000, E1  +396.596, E3 -167593.598}
SPL {X  -159.990, Y  +418.631, Z    +0.000, E1  +410.627, E3 -167596.545}
SPL {X  -159.990, Y  +468.459, Z    +0.000, E1  +425.348, E3 -167616.088}
SPL {X  -159.990, Y  +601.948, Z    +0.000, E1  +428.261, E3 -167702.214}
SPL {X  -159.990, Y  +619.726, Z    +0.000, E1  +428.262, E3 -167717.275}
SPL {X  -159.990, Y  +636.530, Z    +0.000, E1  +428.257, E3 -167731.511}
SPL {X  -159.990, Y  +648.825, Z    +0.000, E1  +428.237, E3 -167741.970}
SPL {X  -159.990, Y  +661.441, Z    +0.000, E1  +428.256, E3 -167752.618}
SPL {X  -159.958, Y  +674.683, Z    +0.000, E1  +428.238, E3 -167763.881}
SPL {X  -159.269, Y  +686.675, Z    +0.000, E1  +428.163, E3 -167774.758}
SPL {X  -157.606, Y  +699.018, Z    +0.000, E1  +427.957, E3 -167786.942}
SPL {X  -155.210, Y  +710.317, Z    +0.000, E1  +427.656, E3 -167798.982}
SPL {X  -152.048, Y  +721.282, Z    +0.000, E1  +427.243, E3 -167811.474}
SPL {X  -148.485, Y  +731.073, Z    +0.000, E1  +426.748, E3 -167823.324}
SPL {X  -145.075, Y  +738.953, Z    +0.000, E1  +426.252, E3 -167833.315}
SPL {X  -141.751, Y  +745.686, Z    +0.000, E1  +425.756, E3 -167842.146}
SPL {X  -138.928, Y  +750.847, Z    +0.000, E1  +425.305, E3 -167849.116}
SPL {X  -136.328, Y  +755.234, Z    +0.000, E1  +424.898, E3 -167855.106}
SPL {X  -132.717, Y  +760.848, Z    +0.000, E1  +424.322, E3 -167862.879}
SPL {X  -128.512, Y  +766.796, Z    +0.000, E1  +423.597, E3 -167871.234}
SPL {X   -99.023, Y  +797.163, Z    +0.000, E1  +413.965, E3 -167973.063}
ENDSPLINE

SPLINE
SPL {X  -130.021, Y  +764.727, Z    +0.000, E1  +405.990, E3 -168112.582}
SPL {X  -148.409, Y  +731.264, Z    +0.000, E1  +396.685, E3 -168136.296}
SPL {X  -155.017, Y  +711.078, Z    +0.000, E1  +387.846, E3 -168143.357}
SPL {X  -158.217, Y  +695.254, Z    +0.000, E1  +378.896, E3 -168146.800}
SPL {X  -159.762, Y  +680.037, Z    +0.000, E1  +368.585, E3 -168148.517}
SPL {X  -159.990, Y  +671.255, Z    +0.000, E1  +361.602, E3 -168148.922}
SPL {X  -159.990, Y  +669.426, Z    +0.000, E1  +359.932, E3 -168148.942}
SPL {X  -159.990, Y  +666.879, Z    +0.000, E1  +356.292, E3 -168148.990}
SPL {X  -159.990, Y  +662.620, Z    +0.000, E1  +348.758, E3 -168149.191}
SPL {X  -159.990, Y  +657.714, Z    +0.000, E1  +339.502, E3 -168149.612}
SPL {X  -159.990, Y  +651.038, Z    +0.000, E1  +327.797, E3 -168150.515}
SPL {X  -159.990, Y  +637.243, Z    +0.000, E1  +311.500, E3 -168153.640}
SPL {X  -159.990, Y  +579.875, Z    +0.000, E1  +294.421, E3 -168176.499}
SPL {X  -159.990, Y  +453.091, Z    +0.000, E1  +291.862, E3 -168259.468}
SPL {X  -159.990, Y  +434.933, Z    +0.000, E1  +291.864, E3 -168274.962}
SPL {X  -159.990, Y  +420.071, Z    +0.000, E1  +291.886, E3 -168287.688}
SPL {X  -159.990, Y  +408.047, Z    +0.000, E1  +291.885, E3 -168297.935}
SPL {X  -159.990, Y  +395.904, Z    +0.000, E1  +291.881, E3 -168308.271}
SPL {X  -157.896, Y  +356.699, Z    +0.000, E1  +289.725, E3 -168320.581}
SPL {X  -156.475, Y  +349.148, Z    +0.000, E1  +290.612, E3 -168334.045}
SPL {X  -155.960, Y  +346.816, Z    +0.000, E1  +291.495, E3 -168343.206}
SPL {X  -154.913, Y  +342.515, Z    +0.000, E1  +292.501, E3 -168355.220}
SPL {X  -152.032, Y  +332.668, Z    +0.000, E1  +292.988, E3 -168367.211}
SPL {X  -148.460, Y  +322.864, Z    +0.000, E1  +293.452, E3 -168379.094}
SPL {X  -144.472, Y  +313.764, Z    +0.000, E1  +294.050, E3 -168390.757}
SPL {X  -140.755, Y  +306.442, Z    +0.000, E1  +294.606, E3 -168400.472}
SPL {X  -137.162, Y  +300.138, Z    +0.000, E1  +295.180, E3 -168409.080}
SPL {X  -134.303, Y  +295.555, Z    +0.000, E1  +295.659, E3 -168415.461}
SPL {X  -131.069, Y  +290.753, Z    +0.000, E1  +296.178, E3 -168422.195}
SPL {X  -127.815, Y  +286.271, Z    +0.000, E1  +296.784, E3 -168428.583}
SPL {X   -98.696, Y  +256.580, Z    +0.000, E1  +308.006, E3 -168564.134}
ENDSPLINE

SPLINE
SPL {X  -138.661, Y  +302.689, Z    +0.000, E1  +316.811, E3 -168681.862}
SPL {X  -154.202, Y  +339.857, Z    +0.000, E1  +330.366, E3 -168699.515}
SPL {X  -158.556, Y  +361.128, Z    +0.000, E1  +342.470, E3 -168704.037}
SPL {X  -159.663, Y  +372.278, Z    +0.000, E1  +350.186, E3 -168705.319}
SPL {X  -159.986, Y  +381.388, Z    +0.000, E1  +357.201, E3 -168705.790}
SPL {X  -159.990, Y  +384.492, Z    +0.000, E1  +359.986, E3 -168705.840}
SPL {X  -159.990, Y  +385.649, Z    +0.000, E1  +361.559, E3 -168705.851}
SPL {X  -159.990, Y  +389.563, Z    +0.000, E1  +367.931, E3 -168705.984}
SPL {X  -159.990, Y  +396.421, Z    +0.000, E1  +380.831, E3 -168706.529}
SPL {X  -159.990, Y  +405.629, Z    +0.000, E1  +396.596, E3 -168707.883}
SPL {X  -159.990, Y  +418.631, Z    +0.000, E1  +410.627, E3 -168710.831}
SPL {X  -159.990, Y  +468.459, Z    +0.000, E1  +425.348, E3 -168730.374}
SPL {X  -159.990, Y  +601.948, Z    +0.000, E1  +428.261, E3 -168816.500}
SPL {X  -159.990, Y  +619.726, Z    +0.000, E1  +428.262, E3 -168831.561}
SPL {X  -159.990, Y  +636.530, Z    +0.000, E1  +428.257, E3 -168845.797}
SPL {X  -159.990, Y  +648.825, Z    +0.000, E1  +428.237, E3 -168856.256}
SPL {X  -159.990, Y  +661.441, Z    +0.000, E1  +428.256, E3 -168866.904}
SPL {X  -159.958, Y  +674.683, Z    +0.000, E1  +428.238, E3 -168878.166}
SPL {X  -159.269, Y  +686.675, Z    +0.000, E1  +428.163, E3 -168889.044}
SPL {X  -158.119, Y  +695.895, Z    +0.000, E1  +428.003, E3 -168898.085}
SPL {X  -156.550, Y  +704.498, Z    +0.000, E1  +427.821, E3 -168906.975}
SPL {X  -153.468, Y  +716.715, Z    +0.000, E1  +427.444, E3 -168920.437}
SPL {X  -149.840, Y  +727.578, Z    +0.000, E1  +426.935, E3 -168933.313}
SPL {X  -145.768, Y  +737.444, Z    +0.000, E1  +426.379, E3 -168945.615}
SPL {X  -141.751, Y  +745.686, Z    +0.000, E1  +425.756, E3 -168956.432}
SPL {X  -138.928, Y  +750.847, Z    +0.000, E1  +425.305, E3 -168963.401}
SPL {X  -136.328, Y  +755.234, Z    +0.000, E1  +424.898, E3 -168969.392}
SPL {X  -132.717, Y  +760.848, Z    +0.000, E1  +424.322, E3 -168977.165}
SPL {X  -128.512, Y  +766.796, Z    +0.000, E1  +423.597, E3 -168985.519}
SPL {X   -99.023, Y  +797.163, Z    +0.000, E1  +413.965, E3 -169087.349}
ENDSPLINE

SPLINE
SPL {X  -130.021, Y  +764.727, Z    +0.000, E1  +405.990, E3 -169226.868}
SPL {X  -148.409, Y  +731.264, Z    +0.000, E1  +396.685, E3 -169250.582}
SPL {X  -155.017, Y  +711.078, Z    +0.000, E1  +387.846, E3 -169257.643}
SPL {X  -158.217, Y  +695.254, Z    +0.000, E1  +378.896, E3 -169261.086}
SPL {X  -159.762, Y  +680.037, Z    +0.000, E1  +368.585, E3 -169262.802}
SPL {X  -159.990, Y  +671.255, Z    +0.000, E1  +361.602, E3 -169263.208}
SPL {X  -159.990, Y  +669.426, Z    +0.000, E1  +359.932, E3 -169263.228}
SPL {X  -159.990, Y  +666.879, Z    +0.000, E1  +356.292, E3 -169263.276}
SPL {X  -159.990, Y  +662.620, Z    +0.000, E1  +348.758, E3 -169263.477}
SPL {X  -159.990, Y  +657.714, Z    +0.000, E1  +339.502, E3 -169263.898}
SPL {X  -159.990, Y  +651.038, Z    +0.000, E1  +327.797, E3 -169264.800}
SPL {X  -159.990, Y  +637.243, Z    +0.000, E1  +311.500, E3 -169267.926}
SPL {X  -159.990, Y  +579.875, Z    +0.000, E1  +294.421, E3 -169290.784}
SPL {X  -159.990, Y  +453.091, Z    +0.000, E1  +291.862, E3 -169373.754}
SPL {X  -159.990, Y  +434.933, Z    +0.000, E1  +291.864, E3 -169389.248}
SPL {X  -159.990, Y  +420.071, Z    +0.000, E1  +291.886, E3 -169401.974}
SPL {X  -159.990, Y  +408.047, Z    +0.000, E1  +291.885, E3 -169412.221}
SPL {X  -159.990, Y  +395.904, Z    +0.000, E1  +291.881, E3 -169422.557}
SPL {X  -157.896, Y  +356.699, Z    +0.000, E1  +289.725, E3 -169434.866}
SPL {X  -156.475, Y  +349.148, Z    +0.000, E1  +290.612, E3 -169448.330}
SPL {X  -155.786, Y  +346.063, Z    +0.000, E1  +291.892, E3 -169461.625}
SPL {X  -153.671, Y  +337.981, Z    +0.000, E1  +292.746, E3 -169475.244}
SPL {X  -150.407, Y  +327.960, Z    +0.000, E1  +293.203, E3 -169487.134}
SPL {X  -147.566, Y  +320.686, Z    +0.000, E1  +293.613, E3 -169496.174}
SPL {X  -144.472, Y  +313.764, Z    +0.000, E1  +294.050, E3 -169505.043}
SPL {X  -140.755, Y  +306.442, Z    +0.000, E1  +294.606, E3 -169514.758}
SPL {X  -137.162, Y  +300.138, Z    +0.000, E1  +295.180, E3 -169523.366}
SPL {X  -132.996, Y  +293.568, Z    +0.000, E1  +295.842, E3 -169532.500}
SPL {X  -128.628, Y  +287.360, Z    +0.000, E1  +296.617, E3 -169541.301}
SPL {X   -98.696, Y  +256.580, Z    +0.000, E1  +308.006, E3 -169678.420}
ENDSPLINE

SPLINE
SPL {X  -138.661, Y  +302.689, Z    +0.000, E1  +316.811, E3 -169796.148}
SPL {X  -154.202, Y  +339.857, Z    +0.000, E1  +330.366, E3 -169813.801}
SPL {X  -158.556, Y  +361.128, Z    +0.000, E1  +342.470, E3 -169818.323}
SPL {X  -159.866, Y  +376.206, Z    +0.000, E1  +353.031, E3 -169819.852}
SPL {X  -159.990, Y  +384.326, Z    +0.000, E1  +359.760, E3 -169820.125}
SPL {X  -159.990, Y  +385.649, Z    +0.000, E1  +361.559, E3 -169820.137}
SPL {X  -159.990, Y  +388.306, Z    +0.000, E1  +365.901, E3 -169820.208}
SPL {X  -159.990, Y  +392.624, Z    +0.000, E1  +373.655, E3 -169820.458}
SPL {X  -159.990, Y  +398.511, Z    +0.000, E1  +384.979, E3 -169821.038}
SPL {X  -159.990, Y  +405.629, Z    +0.000, E1  +396.596, E3 -169822.169}
SPL {X  -159.990, Y  +418.631, Z    +0.000, E1  +410.627, E3 -169825.116}
SPL {X  -159.990, Y  +468.459, Z    +0.000, E1  +425.348, E3 -169844.660}
SPL {X  -159.990, Y  +601.948, Z    +0.000, E1  +428.261, E3 -169930.786}
SPL {X  -159.990, Y  +614.867, Z    +0.000, E1  +428.239, E3 -169941.784}
SPL {X  -159.990, Y  +627.954, Z    +0.000, E1  +428.256, E3 -169952.829}
SPL {X  -159.990, Y  +640.176, Z    +0.000, E1  +428.239, E3 -169963.207}
SPL {X  -159.990, Y  +653.116, Z    +0.000, E1  +428.255, E3 -169974.139}
SPL {X  -159.990, Y  +665.424, Z    +0.000, E1  +428.236, E3 -169984.603}
SPL {X  -159.958, Y  +674.683, Z    +0.000, E1  +428.238, E3 -169992.452}
SPL {X  -159.269, Y  +686.675, Z    +0.000, E1  +428.163, E3 -170003.330}
SPL {X  -158.119, Y  +695.895, Z    +0.000, E1  +428.003, E3 -170012.370}
SPL {X  -156.550, Y  +704.498, Z    +0.000, E1  +427.821, E3 -170021.261}
SPL {X  -153.468, Y  +716.715, Z    +0.000, E1  +427.444, E3 -170034.723}
SPL {X  -149.840, Y  +727.578, Z    +0.000, E1  +426.935, E3 -170047.599}
SPL {X  -145.768, Y  +737.444, Z    +0.000, E1  +426.379, E3 -170059.901}
SPL {X  -141.751, Y  +745.686, Z    +0.000, E1  +425.756, E3 -170070.718}
SPL {X  -138.928, Y  +750.847, Z    +0.000, E1  +425.305, E3 -170077.687}
SPL {X  -136.328, Y  +755.234, Z    +0.000, E1  +424.898, E3 -170083.677}
SPL {X  -132.717, Y  +760.848, Z    +0.000, E1  +424.322, E3 -170091.450}
SPL {X  -128.512, Y  +766.796, Z    +0.000, E1  +423.597, E3 -170099.805}
SPL {X   -99.023, Y  +797.163, Z    +0.000, E1  +413.965, E3 -170201.635}
ENDSPLINE

SPLINE
SPL {X  -130.021, Y  +764.727, Z    +0.000, E1  +405.990, E3 -170341.154}
SPL {X  -148.409, Y  +731.264, Z    +0.000, E1  +396.685, E3 -170364.867}
SPL {X  -155.017, Y  +711.078, Z    +0.000, E1  +387.846, E3 -170371.928}
SPL {X  -158.217, Y  +695.254, Z    +0.000, E1  +378.896, E3 -170375.371}
SPL {X  -159.762, Y  +680.037, Z    +0.000, E1  +368.585, E3 -170377.088}
SPL {X  -159.990, Y  +669.745, Z    +0.000, E1  +360.389, E3 -170377.510}
SPL {X  -159.990, Y  +666.879, Z    +0.000, E1  +356.292, E3 -170377.561}
SPL {X  -159.990, Y  +662.620, Z    +0.000, E1  +348.758, E3 -170377.762}
SPL {X  -159.990, Y  +657.714, Z    +0.000, E1  +339.502, E3 -170378.184}
SPL {X  -159.990, Y  +651.038, Z    +0.000, E1  +327.797, E3 -170379.086}
SPL {X  -159.990, Y  +637.243, Z    +0.000, E1  +311.500, E3 -170382.211}
SPL {X  -159.990, Y  +579.875, Z    +0.000, E1  +294.421, E3 -170405.070}
SPL {X  -159.990, Y  +453.091, Z    +0.000, E1  +291.862, E3 -170488.039}
SPL {X  -159.990, Y  +439.299, Z    +0.000, E1  +291.885, E3 -170499.852}
SPL {X  -159.990, Y  +424.060, Z    +0.000, E1  +291.860, E3 -170512.800}
SPL {X  -159.990, Y  +408.047, Z    +0.000, E1  +291.885, E3 -170526.507}
SPL {X  -159.990, Y  +395.904, Z    +0.000, E1  +291.881, E3 -170536.843}
SPL {X  -157.896, Y  +356.699, Z    +0.000, E1  +289.725, E3 -170549.152}
SPL {X  -156.475, Y  +349.148, Z    +0.000, E1  +290.612, E3 -170562.616}
SPL {X  -155.960, Y  +346.816, Z    +0.000, E1  +291.495, E3 -170571.777}
SPL {X  -154.913, Y  +342.515, Z    +0.000, E1  +292.501, E3 -170583.791}
SPL {X  -152.032, Y  +332.668, Z    +0.000, E1  +292.988, E3 -170595.783}
SPL {X  -149.782, Y  +326.266, Z    +0.000, E1  +293.308, E3 -170603.523}
SPL {X  -146.798, Y  +318.884, Z    +0.000, E1  +293.699, E3 -170612.703}
SPL {X  -143.755, Y  +312.276, Z    +0.000, E1  +294.175, E3 -170621.313}
SPL {X  -140.755, Y  +306.442, Z    +0.000, E1  +294.606, E3 -170629.044}
SPL {X  -137.162, Y  +300.138, Z    +0.000, E1  +295.180, E3 -170637.652}
SPL {X  -134.303, Y  +295.555, Z    +0.000, E1  +295.659, E3 -170644.033}
SPL {X  -132.067, Y  +292.194, Z    +0.000, E1  +296.034, E3 -170648.764}
SPL {X  -128.628, Y  +287.360, Z    +0.000, E1  +296.617, E3 -170655.587}
SPL {X   -99.903, Y  +257.535, Z    +0.000, E1  +308.539, E3 -170804.450}
ENDSPLINE

SPLINE
SPL {X  -141.433, Y  +307.709, Z    +0.000, E1  +318.157, E3 -170914.247}
SPL {X  -151.246, Y  +330.333, Z    +0.000, E1  +326.099, E3 -170925.138}
SPL {X  -155.793, Y  +346.095, Z    +0.000, E1  +333.603, E3 -170929.796}
SPL {X  -158.556, Y  +361.128, Z    +0.000, E1  +342.470, E3 -170932.609}
SPL {X  -159.663, Y  +372.278, Z    +0.000, E1  +350.186, E3 -170933.890}
SPL {X  -159.986, Y  +381.388, Z    +0.000, E1  +357.201, E3 -170934.361}
SPL {X  -159.990, Y  +384.492, Z    +0.000, E1  +359.986, E3 -170934.411}
SPL {X  -159.990, Y  +385.649, Z    +0.000, E1  +361.559, E3 -170934.423}
SPL {X  -159.990, Y  +388.306, Z    +0.000, E1  +365.901, E3 -170934.494}
SPL {X  -159.990, Y  +392.624, Z    +0.000, E1  +373.655, E3 -170934.744}
SPL {X  -159.990, Y  +398.511, Z    +0.000, E1  +384.979, E3 -170935.324}
SPL {X  -159.990, Y  +405.629, Z    +0.000, E1  +396.596, E3 -170936.455}
SPL {X  -159.990, Y  +418.631, Z    +0.000, E1  +410.627, E3 -170939.402}
SPL {X  -159.990, Y  +468.459, Z    +0.000, E1  +425.348, E3 -170958.945}
SPL {X  -159.990, Y  +601.948, Z    +0.000, E1  +428.261, E3 -171045.071}
SPL {X  -159.990, Y  +614.867, Z    +0.000, E1  +428.239, E3 -171056.070}
SPL {X  -159.990, Y  +627.954, Z    +0.000, E1  +428.256, E3 -171067.114}
SPL {X  -159.990, Y  +640.176, Z    +0.000, E1  +428.239, E3 -171077.493}
SPL {X  -159.990, Y  +653.116, Z    +0.000, E1  +428.255, E3 -171088.425}
SPL {X  -159.990, Y  +670.874, Z    +0.000, E1  +428.264, E3 -171103.440}
SPL {X  -159.269, Y  +686.675, Z    +0.000, E1  +428.163, E3 -171117.615}
SPL {X  -158.119, Y  +695.895, Z    +0.000, E1  +428.003, E3 -171126.656}
SPL {X  -156.550, Y  +704.498, Z    +0.000, E1  +427.821, E3 -171135.546}
SPL {X  -154.561, Y  +712.826, Z    +0.000, E1  +427.549, E3 -171144.677}
SPL {X  -152.048, Y  +721.282, Z    +0.000, E1  +427.243, E3 -171154.332}
SPL {X  -148.485, Y  +731.073, Z    +0.000, E1  +426.748, E3 -171166.181}
SPL {X  -145.075, Y  +738.953, Z    +0.000, E1  +426.252, E3 -171176.172}
SPL {X  -141.751, Y  +745.686, Z    +0.000, E1  +425.756, E3 -171185.003}
SPL {X  -138.928, Y  +750.847, Z    +0.000, E1  +425.305, E3 -171191.973}
SPL {X  -136.328, Y  +755.234, Z    +0.000, E1  +424.898, E3 -171197.963}
SPL {X  -132.717, Y  +760.848, Z    +0.000, E1  +424.322, E3 -171205.736}
SPL {X  -128.512, Y  +766.796, Z    +0.000, E1  +423.597, E3 -171214.091}
SPL {X   -99.023, Y  +797.163, Z    +0.000, E1  +413.965, E3 -171315.920}
ENDSPLINE

SPLINE
SPL {X  -130.021, Y  +764.727, Z    +0.000, E1  +405.990, E3 -171455.440}
SPL {X  -148.409, Y  +731.264, Z    +0.000, E1  +396.685, E3 -171479.153}
SPL {X  -155.017, Y  +711.078, Z    +0.000, E1  +387.846, E3 -171486.214}
SPL {X  -158.217, Y  +695.254, Z    +0.000, E1  +378.896, E3 -171489.657}
SPL {X  -159.762, Y  +680.037, Z    +0.000, E1  +368.585, E3 -171491.374}
SPL {X  -159.990, Y  +669.745, Z    +0.000, E1  +360.389, E3 -171491.796}
SPL {X  -159.990, Y  +666.879, Z    +0.000, E1  +356.292, E3 -171491.847}
SPL {X  -159.990, Y  +662.620, Z    +0.000, E1  +348.758, E3 -171492.048}
SPL {X  -159.990, Y  +657.714, Z    +0.000, E1  +339.502, E3 -171492.469}
SPL {X  -159.990, Y  +651.038, Z    +0.000, E1  +327.797, E3 -171493.372}
SPL {X  -159.990, Y  +637.243, Z    +0.000, E1  +311.500, E3 -171496.497}
SPL {X  -159.990, Y  +579.875, Z    +0.000, E1  +294.421, E3 -171519.356}
SPL {X  -159.990, Y  +453.091, Z    +0.000, E1  +291.862, E3 -171602.325}
SPL {X  -159.990, Y  +434.933, Z    +0.000, E1  +291.864, E3 -171617.819}
SPL {X  -159.990, Y  +420.071, Z    +0.000, E1  +291.886, E3 -171630.545}
SPL {X  -159.990, Y  +408.047, Z    +0.000, E1  +291.885, E3 -171640.792}
SPL {X  -159.990, Y  +395.904, Z    +0.000, E1  +291.881, E3 -171651.128}
SPL {X  -157.896, Y  +356.699, Z    +0.000, E1  +289.725, E3 -171663.438}
SPL {X  -156.475, Y  +349.148, Z    +0.000, E1  +290.612, E3 -171676.902}
SPL {X  -155.960, Y  +346.816, Z    +0.000, E1  +291.495, E3 -171686.063}
SPL {X  -154.913, Y  +342.515, Z    +0.000, E1  +292.501, E3 -171698.077}
SPL {X  -152.032, Y  +332.668, Z    +0.000, E1  +292.988, E3 -171710.069}
SPL {X  -148.460, Y  +322.864, Z    +0.000, E1  +293.452, E3 -171721.951}
SPL {X  -144.472, Y  +313.764, Z    +0.000, E1  +294.050, E3 -171733.615}
SPL {X  -141.765, Y  +308.342, Z    +0.000, E1  +294.475, E3 -171740.812}
SPL {X  -139.838, Y  +304.768, Z    +0.000, E1  +294.773, E3 -171745.631}
SPL {X  -137.162, Y  +300.138, Z    +0.000, E1  +295.180, E3 -171751.937}
SPL {X  -132.996, Y  +293.568, Z    +0.000, E1  +295.842, E3 -171761.072}
SPL {X  -128.628, Y  +287.360, Z    +0.000, E1  +296.617, E3 -171769.873}
SPL {X   -99.903, Y  +257.535, Z    +0.000, E1  +308.539, E3 -171918.736}
ENDSPLINE

SPLINE
SPL {X  -141.433, Y  +307.709, Z    +0.000, E1  +318.157, E3 -172028.533}
SPL {X  -151.246, Y  +330.333, Z    +0.000, E1  +326.099, E3 -172039.424}
SPL {X  -155.793, Y  +346.095, Z    +0.000, E1  +333.603, E3 -172044.082}
SPL {X  -158.556, Y  +361.128, Z    +0.000, E1  +342.470, E3 -172046.894}
SPL {X  -159.663, Y  +372.278, Z    +0.000, E1  +350.186, E3 -172048.176}
SPL {X  -159.986, Y  +381.388, Z    +0.000, E1  +357.201, E3 -172048.647}
SPL {X  -159.990, Y  +384.492, Z    +0.000, E1  +359.986, E3 -172048.697}
SPL {X  -159.990, Y  +385.649, Z    +0.000, E1  +361.559, E3 -172048.709}
SPL {X  -159.990, Y  +389.563, Z    +0.000, E1  +367.931, E3 -172048.841}
SPL {X  -159.990, Y  +396.421, Z    +0.000, E1  +380.831, E3 -172049.386}
SPL {X  -159.990, Y  +405.629, Z    +0.000, E1  +396.596, E3 -172050.740}
SPL {X  -159.990, Y  +418.631, Z    +0.000, E1  +410.627, E3 -172053.688}
SPL {X  -159.990, Y  +468.459, Z    +0.000, E1  +425.348, E3 -172073.231}
SPL {X  -159.990, Y  +601.948, Z    +0.000, E1  +428.261, E3 -172159.357}
SPL {X  -159.990, Y  +614.867, Z    +0.000, E1  +428.239, E3 -172170.356}
SPL {X  -159.990, Y  +627.954, Z    +0.000, E1  +428.256, E3 -172181.400}
SPL {X  -159.990, Y  +640.176, Z    +0.000, E1  +428.239, E3 -172191.779}
SPL {X  -159.990, Y  +653.116, Z    +0.000, E1  +428.255, E3 -172202.710}
SPL {X  -159.990, Y  +665.424, Z    +0.000, E1  +428.236, E3 -172213.175}
SPL {X  -159.958, Y  +674.683, Z    +0.000, E1  +428.238, E3 -172221.024}
SPL {X  -159.269, Y  +686.675, Z    +0.000, E1  +428.163, E3 -172231.901}
SPL {X  -158.119, Y  +695.895, Z    +0.000, E1  +428.003, E3 -172240.942}
SPL {X  -156.550, Y  +704.498, Z    +0.000, E1  +427.821, E3 -172249.832}
SPL {X  -153.468, Y  +716.715, Z    +0.000, E1  +427.444, E3 -172263.295}
SPL {X  -149.840, Y  +727.578, Z    +0.000, E1  +426.935, E3 -172276.170}
SPL {X  -145.768, Y  +737.444, Z    +0.000, E1  +426.379, E3 -172288.472}
SPL {X  -141.751, Y  +745.686, Z    +0.000, E1  +425.756, E3 -172299.289}
SPL {X  -138.928, Y  +750.847, Z    +0.000, E1  +425.305, E3 -172306.258}
SPL {X  -136.328, Y  +755.234, Z    +0.000, E1  +424.898, E3 -172312.249}
SPL {X  -132.717, Y  +760.848, Z    +0.000, E1  +424.322, E3 -172320.022}
SPL {X  -128.512, Y  +766.796, Z    +0.000, E1  +423.597, E3 -172328.376}
SPL {X   -99.023, Y  +797.163, Z    +0.000, E1  +413.965, E3 -172430.206}
ENDSPLINE

SPLINE
SPL {X  -130.021, Y  +764.727, Z    +0.000, E1  +405.990, E3 -172569.725}
SPL {X  -148.409, Y  +731.264, Z    +0.000, E1  +396.685, E3 -172593.439}
SPL {X  -155.017, Y  +711.078, Z    +0.000, E1  +387.846, E3 -172600.500}
SPL {X  -158.217, Y  +695.254, Z    +0.000, E1  +378.896, E3 -172603.943}
SPL {X  -159.524, Y  +683.703, Z    +0.000, E1  +371.166, E3 -172605.385}
SPL {X  -159.986, Y  +672.621, Z    +0.000, E1  +362.847, E3 -172606.026}
SPL {X  -159.990, Y  +669.426, Z    +0.000, E1  +359.932, E3 -172606.085}
SPL {X  -159.990, Y  +666.879, Z    +0.000, E1  +356.292, E3 -172606.133}
SPL {X  -159.990, Y  +662.620, Z    +0.000, E1  +348.758, E3 -172606.334}
SPL {X  -159.990, Y  +657.714, Z    +0.000, E1  +339.502, E3 -172606.755}
SPL {X  -159.990, Y  +651.038, Z    +0.000, E1  +327.797, E3 -172607.658}
SPL {X  -159.990, Y  +637.243, Z    +0.000, E1  +311.500, E3 -172610.783}
SPL {X  -159.990, Y  +579.875, Z    +0.000, E1  +294.421, E3 -172633.641}
SPL {X  -159.990, Y  +453.091, Z    +0.000, E1  +291.862, E3 -172716.611}
SPL {X  -159.990, Y  +434.933, Z    +0.000, E1  +291.864, E3 -172732.105}
SPL {X  -159.990, Y  +420.071, Z    +0.000, E1  +291.886, E3 -172744.831}
SPL {X  -159.990, Y  +408.047, Z    +0.000, E1  +291.885, E3 -172755.078}
SPL {X  -159.990, Y  +395.904, Z    +0.000, E1  +291.881, E3 -172765.414}
SPL {X  -157.896, Y  +356.699, Z    +0.000, E1  +289.725, E3 -172777.724}
SPL {X  -156.475, Y  +349.148, Z    +0.000, E1  +290.612, E3 -172791.188}
SPL {X  -155.960, Y  +346.816, Z    +0.000, E1  +291.495, E3 -172800.349}
SPL {X  -154.913, Y  +342.515, Z    +0.000, E1  +292.501, E3 -172812.363}
SPL {X  -152.032, Y  +332.668, Z    +0.000, E1  +292.988, E3 -172824.354}
SPL {X  -149.782, Y  +326.266, Z    +0.000, E1  +293.308, E3 -172832.094}
SPL {X  -146.798, Y  +318.884, Z    +0.000, E1  +293.699, E3 -172841.275}
SPL {X  -143.755, Y  +312.276, Z    +0.000, E1  +294.175, E3 -172849.884}
SPL {X  -140.755, Y  +306.442, Z    +0.000, E1  +294.606, E3 -172857.615}
SPL {X  -137.162, Y  +300.138, Z    +0.000, E1  +295.180, E3 -172866.223}
SPL {X  -134.303, Y  +295.555, Z    +0.000, E1  +295.659, E3 -172872.604}
SPL {X  -132.067, Y  +292.194, Z    +0.000, E1  +296.034, E3 -172877.336}
SPL {X  -128.628, Y  +287.360, Z    +0.000, E1  +296.617, E3 -172884.159}
SPL {X   -99.903, Y  +257.535, Z    +0.000, E1  +308.539, E3 -173033.021}
ENDSPLINE

SPLINE
SPL {X  -141.433, Y  +307.709, Z    +0.000, E1  +318.157, E3 -173142.819}
SPL {X  -151.246, Y  +330.333, Z    +0.000, E1  +326.099, E3 -173153.709}
SPL {X  -155.793, Y  +346.095, Z    +0.000, E1  +333.603, E3 -173158.368}
SPL {X  -158.556, Y  +361.128, Z    +0.000, E1  +342.470, E3 -173161.180}
SPL {X  -159.866, Y  +376.206, Z    +0.000, E1  +353.031, E3 -173162.709}
SPL {X  -159.990, Y  +384.326, Z    +0.000, E1  +359.760, E3 -173162.982}
SPL {X  -159.990, Y  +385.649, Z    +0.000, E1  +361.559, E3 -173162.994}
SPL {X  -159.990, Y  +389.563, Z    +0.000, E1  +367.931, E3 -173163.127}
SPL {X  -159.990, Y  +396.421, Z    +0.000, E1  +380.831, E3 -173163.672}
SPL {X  -159.990, Y  +405.629, Z    +0.000, E1  +396.596, E3 -173165.026}
SPL {X  -159.990, Y  +418.631, Z    +0.000, E1  +410.627, E3 -173167.973}
SPL {X  -159.990, Y  +468.459, Z    +0.000, E1  +425.348, E3 -173187.517}
SPL {X  -159.990, Y  +601.948, Z    +0.000, E1  +428.261, E3 -173273.643}
SPL {X  -159.990, Y  +619.726, Z    +0.000, E1  +428.262, E3 -173288.704}
SPL {X  -159.990, Y  +636.530, Z    +0.000, E1  +428.257, E3 -173302.940}
SPL {X  -159.990, Y  +653.116, Z    +0.000, E1  +428.255, E3 -173316.996}
SPL {X  -159.990, Y  +670.874, Z    +0.000, E1  +428.264, E3 -173332.011}
SPL {X  -159.269, Y  +686.675, Z    +0.000, E1  +428.163, E3 -173346.187}
SPL {X  -158.119, Y  +695.895, Z    +0.000, E1  +428.003, E3 -173355.227}
SPL {X  -156.550, Y  +704.498, Z    +0.000, E1  +427.821, E3 -173364.118}
SPL {X  -154.561, Y  +712.826, Z    +0.000, E1  +427.549, E3 -173373.248}
SPL {X  -152.048, Y  +721.282, Z    +0.000, E1  +427.243, E3 -173382.903}
SPL {X  -148.485, Y  +731.073, Z    +0.000, E1  +426.748, E3 -173394.752}
SPL {X  -145.075, Y  +738.953, Z    +0.000, E1  +426.252, E3 -173404.744}
SPL {X  -141.751, Y  +745.686, Z    +0.000, E1  +425.756, E3 -173413.575}
SPL {X  -138.928, Y  +750.847, Z    +0.000, E1  +425.305, E3 -173420.544}
SPL {X  -136.328, Y  +755.234, Z    +0.000, E1  +424.898, E3 -173426.534}
SPL {X  -132.717, Y  +760.848, Z    +0.000, E1  +424.322, E3 -173434.308}
SPL {X  -128.512, Y  +766.796, Z    +0.000, E1  +423.597, E3 -173442.662}
SPL {X   -99.023, Y  +797.163, Z    +0.000, E1  +413.965, E3 -173544.492}
ENDSPLINE

SPLINE
SPL {X  -130.021, Y  +764.727, Z    +0.000, E1  +405.990, E3 -173684.011}
SPL {X  -148.409, Y  +731.264, Z    +0.000, E1  +396.685, E3 -173707.725}
SPL {X  -155.017, Y  +711.078, Z    +0.000, E1  +387.846, E3 -173714.786}
SPL {X  -158.217, Y  +695.254, Z    +0.000, E1  +378.896, E3 -173718.228}
SPL {X  -159.762, Y  +680.037, Z    +0.000, E1  +368.585, E3 -173719.945}
SPL {X  -159.990, Y  +671.255, Z    +0.000, E1  +361.602, E3 -173720.351}
SPL {X  -159.990, Y  +669.426, Z    +0.000, E1  +359.932, E3 -173720.371}
SPL {X  -159.990, Y  +666.879, Z    +0.000, E1  +356.292, E3 -173720.418}
SPL {X  -159.990, Y  +662.620, Z    +0.000, E1  +348.758, E3 -173720.620}
SPL {X  -159.990, Y  +657.714, Z    +0.000, E1  +339.502, E3 -173721.041}
SPL {X  -159.990, Y  +651.038, Z    +0.000, E1  +327.797, E3 -173721.943}
SPL {X  -159.990, Y  +637.243, Z    +0.000, E1  +311.500, E3 -173725.068}
SPL {X  -159.990, Y  +579.875, Z    +0.000, E1  +294.421, E3 -173747.927}
SPL {X  -159.990, Y  +453.091, Z    +0.000, E1  +291.862, E3 -173830.897}
SPL {X  -159.990, Y  +434.933, Z    +0.000, E1  +291.864, E3 -173846.390}
SPL {X  -159.990, Y  +420.071, Z    +0.000, E1  +291.886, E3 -173859.116}
SPL {X  -159.990, Y  +408.047, Z    +0.000, E1  +291.885, E3 -173869.364}
SPL {X  -159.990, Y  +395.904, Z    +0.000, E1  +291.881, E3 -173879.700}
SPL {X  -158.518, Y  +360.846, Z    +0.000, E1  +289.610, E3 -173887.635}
SPL {X  -157.390, Y  +353.775, Z    +0.000, E1  +289.868, E3 -173895.311}
SPL {X  -156.475, Y  +349.148, Z    +0.000, E1  +290.612, E3 -173905.473}
SPL {X  -155.960, Y  +346.816, Z    +0.000, E1  +291.495, E3 -173914.635}
SPL {X  -154.913, Y  +342.515, Z    +0.000, E1  +292.501, E3 -173926.649}
SPL {X  -152.032, Y  +332.668, Z    +0.000, E1  +292.988, E3 -173938.640}
SPL {X  -149.782, Y  +326.266, Z    +0.000, E1  +293.308, E3 -173946.380}
SPL {X  -146.798, Y  +318.884, Z    +0.000, E1  +293.699, E3 -173955.561}
SPL {X  -143.755, Y  +312.276, Z    +0.000, E1  +294.175, E3 -173964.170}
SPL {X  -140.755, Y  +306.442, Z    +0.000, E1  +294.606, E3 -173971.901}
SPL {X  -137.162, Y  +300.138, Z    +0.000, E1  +295.180, E3 -173980.509}
SPL {X  -134.303, Y  +295.555, Z    +0.000, E1  +295.659, E3 -173986.890}
SPL {X  -132.067, Y  +292.194, Z    +0.000, E1  +296.034, E3 -173991.621}
SPL {X  -128.628, Y  +287.360, Z    +0.000, E1  +296.617, E3 -173998.444}
SPL {X   -98.696, Y  +256.580, Z    +0.000, E1  +308.006, E3 -174135.562}
ENDSPLINE

SPLINE
SPL {X  -138.661, Y  +302.689, Z    +0.000, E1  +316.811, E3 -174253.291}
SPL {X  -154.202, Y  +339.857, Z    +0.000, E1  +330.366, E3 -174270.944}
SPL {X  -158.556, Y  +361.128, Z    +0.000, E1  +342.470, E3 -174275.466}
SPL {X  -159.866, Y  +376.206, Z    +0.000, E1  +353.031, E3 -174276.995}
SPL {X  -159.990, Y  +384.789, Z    +0.000, E1  +360.146, E3 -174277.272}
SPL {X  -159.990, Y  +388.306, Z    +0.000, E1  +365.901, E3 -174277.351}
SPL {X  -159.990, Y  +392.624, Z    +0.000, E1  +373.655, E3 -174277.601}
SPL {X  -159.990, Y  +398.511, Z    +0.000, E1  +384.979, E3 -174278.181}
SPL {X  -159.990, Y  +405.629, Z    +0.000, E1  +396.596, E3 -174279.312}
SPL {X  -159.990, Y  +418.631, Z    +0.000, E1  +410.627, E3 -174282.259}
SPL {X  -159.990, Y  +468.459, Z    +0.000, E1  +425.348, E3 -174301.803}
SPL {X  -159.990, Y  +601.948, Z    +0.000, E1  +428.261, E3 -174387.929}
SPL {X  -159.990, Y  +614.867, Z    +0.000, E1  +428.239, E3 -174398.927}
SPL {X  -159.990, Y  +627.954, Z    +0.000, E1  +428.256, E3 -174409.971}
SPL {X  -159.990, Y  +640.176, Z    +0.000, E1  +428.239, E3 -174420.350}
SPL {X  -159.990, Y  +653.116, Z    +0.000, E1  +428.255, E3 -174431.282}
SPL {X  -159.990, Y  +665.424, Z    +0.000, E1  +428.236, E3 -174441.746}
SPL {X  -159.958, Y  +674.683, Z    +0.000, E1  +428.238, E3 -174449.595}
SPL {X  -159.269, Y  +686.675, Z    +0.000, E1  +428.163, E3 -174460.472}
SPL {X  -157.606, Y  +699.018, Z    +0.000, E1  +427.957, E3 -174472.656}
SPL {X  -155.210, Y  +710.317, Z    +0.000, E1  +427.656, E3 -174484.696}
SPL {X  -152.683, Y  +719.299, Z    +0.000, E1  +427.307, E3 -174494.908}
SPL {X  -149.840, Y  +727.578, Z    +0.000, E1  +426.935, E3 -174504.742}
SPL {X  -145.768, Y  +737.444, Z    +0.000, E1  +426.379, E3 -174517.044}
SPL {X  -141.751, Y  +745.686, Z    +0.000, E1  +425.756, E3 -174527.860}
SPL {X  -138.928, Y  +750.847, Z    +0.000, E1  +425.305, E3 -174534.830}
SPL {X  -136.328, Y  +755.234, Z    +0.000, E1  +424.898, E3 -174540.820}
SPL {X  -132.717, Y  +760.848, Z    +0.000, E1  +424.322, E3 -174548.593}
SPL {X  -129.778, Y  +765.065, Z    +0.000, E1  +423.787, E3 -174554.548}
SPL {X  -127.600, Y  +768.014, Z    +0.000, E1  +423.408, E3 -174558.695}
SPL {X   -99.023, Y  +797.163, Z    +0.000, E1  +413.965, E3 -174658.777}
ENDSPLINE

SPLINE
SPL {X  -130.021, Y  +764.727, Z    +0.000, E1  +405.990, E3 -174798.297}
SPL {X  -148.409, Y  +731.264, Z    +0.000, E1  +396.685, E3 -174822.010}
SPL {X  -155.017, Y  +711.078, Z    +0.000, E1  +387.846, E3 -174829.071}
SPL {X  -158.217, Y  +695.254, Z    +0.000, E1  +378.896, E3 -174832.514}
SPL {X  -159.524, Y  +683.703, Z    +0.000, E1  +371.166, E3 -174833.956}
SPL {X  -159.986, Y  +672.621, Z    +0.000, E1  +362.847, E3 -174834.598}
SPL {X  -159.990, Y  +669.148, Z    +0.000, E1  +359.679, E3 -174834.659}
SPL {X  -159.990, Y  +666.130, Z    +0.000, E1  +354.946, E3 -174834.725}
SPL {X  -159.990, Y  +662.620, Z    +0.000, E1  +348.758, E3 -174834.905}
SPL {X  -159.990, Y  +657.714, Z    +0.000, E1  +339.502, E3 -174835.327}
SPL {X  -159.990, Y  +651.038, Z    +0.000, E1  +327.797, E3 -174836.229}
SPL {X  -159.990, Y  +637.243, Z    +0.000, E1  +311.500, E3 -174839.354}
SPL {X  -159.990, Y  +579.875, Z    +0.000, E1  +294.421, E3 -174862.213}
SPL {X  -159.990, Y  +453.091, Z    +0.000, E1  +291.862, E3 -174945.182}
SPL {X  -159.990, Y  +434.933, Z    +0.000, E1  +291.864, E3 -174960.676}
SPL {X  -159.990, Y  +420.071, Z    +0.000, E1  +291.886, E3 -174973.402}
SPL {X  -159.990, Y  +408.047, Z    +0.000, E1  +291.885, E3 -174983.650}
SPL {X  -159.990, Y  +395.904, Z    +0.000, E1  +291.881, E3 -174993.986}
SPL {X  -157.896, Y  +356.699, Z    +0.000, E1  +289.725, E3 -175006.295}
SPL {X  -156.475, Y  +349.148, Z    +0.000, E1  +290.612, E3 -175019.759}
SPL {X  -155.786, Y  +346.063, Z    +0.000, E1  +291.892, E3 -175033.053}
SPL {X  -154.401, Y  +340.583, Z    +0.000, E1  +292.675, E3 -175043.750}
SPL {X  -152.032, Y  +332.668, Z    +0.000, E1  +292.988, E3 -175052.926}
SPL {X  -148.460, Y  +322.864, Z    +0.000, E1  +293.452, E3 -175064.808}
SPL {X  -144.472, Y  +313.764, Z    +0.000, E1  +294.050, E3 -175076.472}
SPL {X  -140.755, Y  +306.442, Z    +0.000, E1  +294.606, E3 -175086.186}
SPL {X  -137.162, Y  +300.138, Z    +0.000, E1  +295.180, E3 -175094.795}
SPL {X  -134.303, Y  +295.555, Z    +0.000, E1  +295.659, E3 -175101.175}
SPL {X  -131.069, Y  +290.753, Z    +0.000, E1  +296.178, E3 -175107.909}
SPL {X  -127.815, Y  +286.271, Z    +0.000, E1  +296.784, E3 -175114.297}
SPL {X   -99.903, Y  +257.535, Z    +0.000, E1  +308.539, E3 -175261.593}
ENDSPLINE

SPLINE
SPL {X  -141.433, Y  +307.709, Z    +0.000, E1  +318.157, E3 -175371.390}
SPL {X  -151.246, Y  +330.333, Z    +0.000, E1  +326.099, E3 -175382.281}
SPL {X  -155.793, Y  +346.095, Z    +0.000, E1  +333.603, E3 -175386.939}
SPL {X  -158.556, Y  +361.128, Z    +0.000, E1  +342.470, E3 -175389.751}
SPL {X  -159.663, Y  +372.278, Z    +0.000, E1  +350.186, E3 -175391.033}
SPL {X  -159.986, Y  +381.388, Z    +0.000, E1  +357.201, E3 -175391.504}
SPL {X  -159.990, Y  +384.492, Z    +0.000, E1  +359.986, E3 -175391.554}
SPL {X  -159.990, Y  +385.649, Z    +0.000, E1  +361.559, E3 -175391.566}
SPL {X  -159.990, Y  +388.306, Z    +0.000, E1  +365.901, E3 -175391.637}
SPL {X  -159.990, Y  +392.624, Z    +0.000, E1  +373.655, E3 -175391.887}
SPL {X  -159.990, Y  +398.511, Z    +0.000, E1  +384.979, E3 -175392.467}
SPL {X  -159.990, Y  +405.629, Z    +0.000, E1  +396.596, E3 -175393.598}
SPL {X  -159.990, Y  +418.631, Z    +0.000, E1  +410.627, E3 -175396.545}
SPL {X  -159.990, Y  +468.459, Z    +0.000, E1  +425.348, E3 -175416.088}
SPL {X  -159.990, Y  +595.966, Z    +0.000, E1  +428.240, E3 -175497.199}
SPL {X  -159.990, Y  +605.502, Z    +0.000, E1  +428.241, E3 -175505.276}
SPL {X  -159.990, Y  +619.726, Z    +0.000, E1  +428.262, E3 -175517.275}
SPL {X  -159.990, Y  +636.530, Z    +0.000, E1  +428.257, E3 -175531.511}
SPL {X  -159.990, Y  +653.116, Z    +0.000, E1  +428.255, E3 -175545.568}
SPL {X  -159.990, Y  +670.874, Z    +0.000, E1  +428.264, E3 -175560.582}
SPL {X  -159.269, Y  +686.675, Z    +0.000, E1  +428.163, E3 -175574.758}
SPL {X  -157.606, Y  +699.018, Z    +0.000, E1  +427.957, E3 -175586.942}
SPL {X  -155.210, Y  +710.317, Z    +0.000, E1  +427.656, E3 -175598.982}
SPL {X  -152.683, Y  +719.299, Z    +0.000, E1  +427.307, E3 -175609.194}
SPL {X  -149.840, Y  +727.578, Z    +0.000, E1  +426.935, E3 -175619.028}
SPL {X  -145.768, Y  +737.444, Z    +0.000, E1  +426.379, E3 -175631.330}
SPL {X  -141.751, Y  +745.686, Z    +0.000, E1  +425.756, E3 -175642.146}
SPL {X  -138.928, Y  +750.847, Z    +0.000, E1  +425.305, E3 -175649.116}
SPL {X  -135.390, Y  +756.743, Z    +0.000, E1  +424.775, E3 -175657.148}
SPL {X  -132.002, Y  +761.900, Z    +0.000, E1  +424.179, E3 -175664.379}
SPL {X  -128.512, Y  +766.796, Z    +0.000, E1  +423.597, E3 -175671.234}
SPL {X   -99.023, Y  +797.163, Z    +0.000, E1  +413.965, E3 -175773.063}
ENDSPLINE

SPLINE
SPL {X  -130.021, Y  +764.727, Z    +0.000, E1  +405.990, E3 -175912.582}
SPL {X  -148.409, Y  +731.264, Z    +0.000, E1  +396.685, E3 -175936.296}
SPL {X  -155.017, Y  +711.078, Z    +0.000, E1  +387.846, E3 -175943.357}
SPL {X  -158.217, Y  +695.254, Z    +0.000, E1  +378.896, E3 -175946.800}
SPL {X  -159.524, Y  +683.703, Z    +0.000, E1  +371.166, E3 -175948.242}
SPL {X  -159.986, Y  +672.621, Z    +0.000, E1  +362.847, E3 -175948.884}
SPL {X  -159.990, Y  +669.148, Z    +0.000, E1  +359.679, E3 -175948.945}
SPL {X  -159.990, Y  +666.130, Z    +0.000, E1  +354.946, E3 -175949.011}
SPL {X  -159.990, Y  +662.620, Z    +0.000, E1  +348.758, E3 -175949.191}
SPL {X  -159.990, Y  +657.714, Z    +0.000, E1  +339.502, E3 -175949.612}
SPL {X  -159.990, Y  +651.038, Z    +0.000, E1  +327.797, E3 -175950.515}
SPL {X  -159.990, Y  +637.243, Z    +0.000, E1  +311.500, E3 -175953.640}
SPL {X  -159.990, Y  +579.875, Z    +0.000, E1  +294.421, E3 -175976.499}
SPL {X  -159.990, Y  +453.091, Z    +0.000, E1  +291.862, E3 -176059.468}
SPL {X  -159.990, Y  +434.933, Z    +0.000, E1  +291.864, E3 -176074.962}
SPL {X  -159.990, Y  +420.071, Z    +0.000, E1  +291.886, E3 -176087.688}
SPL {X  -159.990, Y  +408.047, Z    +0.000, E1  +291.885, E3 -176097.935}
SPL {X  -159.990, Y  +395.904, Z    +0.000, E1  +291.881, E3 -176108.271}
SPL {X  -157.896, Y  +356.699, Z    +0.000, E1  +289.725, E3 -176120.581}
SPL {X  -156.475, Y  +349.148, Z    +0.000, E1  +290.612, E3 -176134.045}
SPL {X  -155.960, Y  +346.816, Z    +0.000, E1  +291.495, E3 -176143.206}
SPL {X  -154.913, Y  +342.515, Z    +0.000, E1  +292.501, E3 -176155.220}
SPL {X  -152.032, Y  +332.668, Z    +0.000, E1  +292.988, E3 -176167.211}
SPL {X  -149.782, Y  +326.266, Z    +0.000, E1  +293.308, E3 -176174.951}
SPL {X  -146.798, Y  +318.884, Z    +0.000, E1  +293.699, E3 -176184.132}
SPL {X  -143.755, Y  +312.276, Z    +0.000, E1  +294.175, E3 -176192.741}
SPL {X  -140.755, Y  +306.442, Z    +0.000, E1  +294.606, E3 -176200.472}
SPL {X  -137.162, Y  +300.138, Z    +0.000, E1  +295.180, E3 -176209.080}
SPL {X  -134.303, Y  +295.555, Z    +0.000, E1  +295.659, E3 -176215.461}
SPL {X  -132.067, Y  +292.194, Z    +0.000, E1  +296.034, E3 -176220.193}
SPL {X  -128.628, Y  +287.360, Z    +0.000, E1  +296.617, E3 -176227.016}
SPL {X   -98.696, Y  +256.580, Z    +0.000, E1  +308.006, E3 -176364.134}
ENDSPLINE

SPLINE
SPL {X  -138.661, Y  +302.689, Z    +0.000, E1  +316.811, E3 -176481.862}
SPL {X  -154.202, Y  +339.857, Z    +0.000, E1  +330.366, E3 -176499.515}
SPL {X  -158.556, Y  +361.128, Z    +0.000, E1  +342.470, E3 -176504.037}
SPL {X  -159.866, Y  +376.206, Z    +0.000, E1  +353.031, E3 -176505.566}
SPL {X  -159.990, Y  +384.326, Z    +0.000, E1  +359.760, E3 -176505.839}
SPL {X  -159.990, Y  +385.649, Z    +0.000, E1  +361.559, E3 -176505.851}
SPL {X  -159.990, Y  +388.306, Z    +0.000, E1  +365.901, E3 -176505.923}
SPL {X  -159.990, Y  +392.624, Z    +0.000, E1  +373.655, E3 -176506.172}
SPL {X  -159.990, Y  +398.511, Z    +0.000, E1  +384.979, E3 -176506.752}
SPL {X  -159.990, Y  +405.629, Z    +0.000, E1  +396.596, E3 -176507.883}
SPL {X  -159.990, Y  +418.631, Z    +0.000, E1  +410.627, E3 -176510.831}
SPL {X  -159.990, Y  +468.459, Z    +0.000, E1  +425.348, E3 -176530.374}
SPL {X  -159.990, Y  +601.948, Z    +0.000, E1  +428.261, E3 -176616.500}
SPL {X  -159.990, Y  +619.726, Z    +0.000, E1  +428.262, E3 -176631.561}
SPL {X  -159.990, Y  +636.530, Z    +0.000, E1  +428.257, E3 -176645.797}
SPL {X  -159.990, Y  +653.116, Z    +0.000, E1  +428.255, E3 -176659.853}
SPL {X  -159.990, Y  +670.874, Z    +0.000, E1  +428.264, E3 -176674.868}
SPL {X  -159.269, Y  +686.675, Z    +0.000, E1  +428.163, E3 -176689.044}
SPL {X  -157.606, Y  +699.018, Z    +0.000, E1  +427.957, E3 -176701.228}
SPL {X  -155.210, Y  +710.317, Z    +0.000, E1  +427.656, E3 -176713.268}
SPL {X  -152.048, Y  +721.282, Z    +0.000, E1  +427.243, E3 -176725.760}
SPL {X  -148.485, Y  +731.073, Z    +0.000, E1  +426.748, E3 -176737.609}
SPL {X  -145.075, Y  +738.953, Z    +0.000, E1  +426.252, E3 -176747.601}
SPL {X  -141.751, Y  +745.686, Z    +0.000, E1  +425.756, E3 -176756.432}
SPL {X  -138.928, Y  +750.847, Z    +0.000, E1  +425.305, E3 -176763.401}
SPL {X  -135.390, Y  +756.743, Z    +0.000, E1  +424.775, E3 -176771.433}
SPL {X  -132.002, Y  +761.900, Z    +0.000, E1  +424.179, E3 -176778.665}
SPL {X  -128.512, Y  +766.796, Z    +0.000, E1  +423.597, E3 -176785.519}
SPL {X   -99.023, Y  +797.163, Z    +0.000, E1  +413.965, E3 -176887.349}
ENDSPLINE

SPLINE
SPL {X  -130.021, Y  +764.727, Z    +0.000, E1  +405.990, E3 -177026.868}
SPL {X  -148.409, Y  +731.264, Z    +0.000, E1  +396.685, E3 -177050.582}
SPL {X  -155.017, Y  +711.078, Z    +0.000, E1  +387.846, E3 -177057.643}
SPL {X  -158.217, Y  +695.254, Z    +0.000, E1  +378.896, E3 -177061.086}
SPL {X  -159.762, Y  +680.037, Z    +0.000, E1  +368.585, E3 -177062.802}
SPL {X  -159.990, Y  +671.255, Z    +0.000, E1  +361.602, E3 -177063.208}
SPL {X  -159.990, Y  +669.148, Z    +0.000, E1  +359.679, E3 -177063.231}
SPL {X  -159.990, Y  +666.130, Z    +0.000, E1  +354.946, E3 -177063.296}
SPL {X  -159.990, Y  +662.620, Z    +0.000, E1  +348.758, E3 -177063.477}
SPL {X  -159.990, Y  +657.714, Z    +0.000, E1  +339.502, E3 -177063.898}
SPL {X  -159.990, Y  +651.038, Z    +0.000, E1  +327.797, E3 -177064.800}
SPL {X  -159.990, Y  +637.243, Z    +0.000, E1  +311.500, E3 -177067.926}
SPL {X  -159.990, Y  +579.875, Z    +0.000, E1  +294.421, E3 -177090.784}
SPL {X  -159.990, Y  +453.091, Z    +0.000, E1  +291.862, E3 -177173.754}
SPL {X  -159.990, Y  +439.299, Z    +0.000, E1  +291.885, E3 -177185.566}
SPL {X  -159.990, Y  +424.060, Z    +0.000, E1  +291.860, E3 -177198.515}
SPL {X  -159.990, Y  +408.047, Z    +0.000, E1  +291.885, E3 -177212.221}
SPL {X  -159.990, Y  +395.904, Z    +0.000, E1  +291.881, E3 -177222.557}
SPL {X  -157.896, Y  +356.699, Z    +0.000, E1  +289.725, E3 -177234.866}
SPL {X  -156.475, Y  +349.148, Z    +0.000, E1  +290.612, E3 -177248.330}
SPL {X  -155.786, Y  +346.063, Z    +0.000, E1  +291.892, E3 -177261.625}
SPL {X  -154.401, Y  +340.583, Z    +0.000, E1  +292.675, E3 -177272.322}
SPL {X  -152.032, Y  +332.668, Z    +0.000, E1  +292.988, E3 -177281.497}
SPL {X  -149.782, Y  +326.266, Z    +0.000, E1  +293.308, E3 -177289.237}
SPL {X  -146.798, Y  +318.884, Z    +0.000, E1  +293.699, E3 -177298.418}
SPL {X  -143.755, Y  +312.276, Z    +0.000, E1  +294.175, E3 -177307.027}
SPL {X  -140.755, Y  +306.442, Z    +0.000, E1  +294.606, E3 -177314.758}
SPL {X  -137.162, Y  +300.138, Z    +0.000, E1  +295.180, E3 -177323.366}
SPL {X  -134.303, Y  +295.555, Z    +0.000, E1  +295.659, E3 -177329.747}
SPL {X  -132.067, Y  +292.194, Z    +0.000, E1  +296.034, E3 -177334.479}
SPL {X  -128.628, Y  +287.360, Z    +0.000, E1  +296.617, E3 -177341.301}
SPL {X   -98.696, Y  +256.580, Z    +0.000, E1  +308.006, E3 -177478.420}
ENDSPLINE

SPLINE
SPL {X  -138.661, Y  +302.689, Z    +0.000, E1  +316.811, E3 -177596.148}
SPL {X  -154.202, Y  +339.857, Z    +0.000, E1  +330.366, E3 -177613.801}
SPL {X  -158.556, Y  +361.128, Z    +0.000, E1  +342.470, E3 -177618.323}
SPL {X  -159.866, Y  +376.206, Z    +0.000, E1  +353.031, E3 -177619.852}
SPL {X  -159.990, Y  +384.326, Z    +0.000, E1  +359.760, E3 -177620.125}
SPL {X  -159.990, Y  +385.649, Z    +0.000, E1  +361.559, E3 -177620.137}
SPL {X  -159.990, Y  +389.563, Z    +0.000, E1  +367.931, E3 -177620.269}
SPL {X  -159.990, Y  +396.421, Z    +0.000, E1  +380.831, E3 -177620.814}
SPL {X  -159.990, Y  +405.629, Z    +0.000, E1  +396.596, E3 -177622.169}
SPL {X  -159.990, Y  +418.631, Z    +0.000, E1  +410.627, E3 -177625.116}
SPL {X  -159.990, Y  +468.459, Z    +0.000, E1  +425.348, E3 -177644.660}
SPL {X  -159.990, Y  +601.948, Z    +0.000, E1  +428.261, E3 -177730.786}
SPL {X  -159.990, Y  +619.726, Z    +0.000, E1  +428.262, E3 -177745.846}
SPL {X  -159.990, Y  +636.530, Z    +0.000, E1  +428.257, E3 -177760.083}
SPL {X  -159.990, Y  +653.116, Z    +0.000, E1  +428.255, E3 -177774.139}
SPL {X  -159.990, Y  +665.424, Z    +0.000, E1  +428.236, E3 -177784.603}
SPL {X  -159.958, Y  +674.683, Z    +0.000, E1  +428.238, E3 -177792.452}
SPL {X  -159.269, Y  +686.675, Z    +0.000, E1  +428.163, E3 -177803.330}
SPL {X  -158.119, Y  +695.895, Z    +0.000, E1  +428.003, E3 -177812.370}
SPL {X  -156.550, Y  +704.498, Z    +0.000, E1  +427.821, E3 -177821.261}
SPL {X  -154.561, Y  +712.826, Z    +0.000, E1  +427.549, E3 -177830.391}
SPL {X  -152.048, Y  +721.282, Z    +0.000, E1  +427.243, E3 -177840.046}
SPL {X  -148.485, Y  +731.073, Z    +0.000, E1  +426.748, E3 -177851.895}
SPL {X  -145.075, Y  +738.953, Z    +0.000, E1  +426.252, E3 -177861.887}
SPL {X  -141.751, Y  +745.686, Z    +0.000, E1  +425.756, E3 -177870.718}
SPL {X  -138.928, Y  +750.847, Z    +0.000, E1  +425.305, E3 -177877.687}
SPL {X  -135.390, Y  +756.743, Z    +0.000, E1  +424.775, E3 -177885.719}
SPL {X  -132.002, Y  +761.900, Z    +0.000, E1  +424.179, E3 -177892.951}
SPL {X  -128.512, Y  +766.796, Z    +0.000, E1  +423.597, E3 -177899.805}
SPL {X   -99.023, Y  +797.163, Z    +0.000, E1  +413.965, E3 -178001.635}
ENDSPLINE

SPLINE
SPL {X  -130.021, Y  +764.727, Z    +0.000, E1  +405.990, E3 -178141.154}
SPL {X  -148.409, Y  +731.264, Z    +0.000, E1  +396.685, E3 -178164.867}
SPL {X  -155.017, Y  +711.078, Z    +0.000, E1  +387.846, E3 -178171.928}
SPL {X  -158.217, Y  +695.254, Z    +0.000, E1  +378.896, E3 -178175.371}
SPL {X  -159.524, Y  +683.703, Z    +0.000, E1  +371.166, E3 -178176.813}
SPL {X  -159.986, Y  +672.621, Z    +0.000, E1  +362.847, E3 -178177.455}
SPL {X  -159.990, Y  +669.148, Z    +0.000, E1  +359.679, E3 -178177.516}
SPL {X  -159.990, Y  +666.130, Z    +0.000, E1  +354.946, E3 -178177.582}
SPL {X  -159.990, Y  +662.620, Z    +0.000, E1  +348.758, E3 -178177.762}
SPL {X  -159.990, Y  +657.714, Z    +0.000, E1  +339.502, E3 -178178.184}
SPL {X  -159.990, Y  +651.038, Z    +0.000, E1  +327.797, E3 -178179.086}
SPL {X  -159.990, Y  +642.324, Z    +0.000, E1  +316.129, E3 -178180.821}
SPL {X  -159.990, Y  +634.003, Z    +0.000, E1  +308.893, E3 -178183.096}
SPL {X  -159.990, Y  +579.875, Z    +0.000, E1  +294.421, E3 -178205.070}
SPL {X  -159.990, Y  +453.091, Z    +0.000, E1  +291.862, E3 -178288.039}
SPL {X  -159.990, Y  +434.933, Z    +0.000, E1  +291.864, E3 -178303.533}
SPL {X  -159.990, Y  +420.071, Z    +0.000, E1  +291.886, E3 -178316.259}
SPL {X  -159.990, Y  +408.047, Z    +0.000, E1  +291.885, E3 -178326.507}
SPL {X  -159.990, Y  +395.904, Z    +0.000, E1  +291.881, E3 -178336.843}
SPL {X  -157.896, Y  +356.699, Z    +0.000, E1  +289.725, E3 -178349.152}
SPL {X  -156.475, Y  +349.148, Z    +0.000, E1  +290.612, E3 -178362.616}
SPL {X  -155.786, Y  +346.063, Z    +0.000, E1  +291.892, E3 -178375.911}
SPL {X  -153.671, Y  +337.981, Z    +0.000, E1  +292.746, E3 -178389.530}
SPL {X  -150.407, Y  +327.960, Z    +0.000, E1  +293.203, E3 -178401.420}
SPL {X  -147.566, Y  +320.686, Z    +0.000, E1  +293.613, E3 -178410.459}
SPL {X  -144.472, Y  +313.764, Z    +0.000, E1  +294.050, E3 -178419.329}
SPL {X  -140.755, Y  +306.442, Z    +0.000, E1  +294.606, E3 -178429.044}
SPL {X  -137.162, Y  +300.138, Z    +0.000, E1  +295.180, E3 -178437.652}
SPL {X  -134.303, Y  +295.555, Z    +0.000, E1  +295.659, E3 -178444.033}
SPL {X  -132.067, Y  +292.194, Z    +0.000, E1  +296.034, E3 -178448.764}
SPL {X  -128.628, Y  +287.360, Z    +0.000, E1  +296.617, E3 -178455.587}
SPL {X   -99.903, Y  +257.535, Z    +0.000, E1  +308.539, E3 -178604.450}
ENDSPLINE

SPLINE
SPL {X  -141.433, Y  +307.709, Z    +0.000, E1  +318.157, E3 -178714.247}
SPL {X  -151.246, Y  +330.333, Z    +0.000, E1  +326.099, E3 -178725.138}
SPL {X  -155.793, Y  +346.095, Z    +0.000, E1  +333.603, E3 -178729.796}
SPL {X  -158.556, Y  +361.128, Z    +0.000, E1  +342.470, E3 -178732.609}
SPL {X  -159.866, Y  +376.206, Z    +0.000, E1  +353.031, E3 -178734.138}
SPL {X  -159.990, Y  +384.789, Z    +0.000, E1  +360.146, E3 -178734.415}
SPL {X  -159.990, Y  +388.306, Z    +0.000, E1  +365.901, E3 -178734.494}
SPL {X  -159.990, Y  +392.624, Z    +0.000, E1  +373.655, E3 -178734.744}
SPL {X  -159.990, Y  +398.511, Z    +0.000, E1  +384.979, E3 -178735.324}
SPL {X  -159.990, Y  +405.629, Z    +0.000, E1  +396.596, E3 -178736.455}
SPL {X  -159.990, Y  +418.631, Z    +0.000, E1  +410.627, E3 -178739.402}
SPL {X  -159.990, Y  +468.459, Z    +0.000, E1  +425.348, E3 -178758.945}
SPL {X  -159.990, Y  +595.966, Z    +0.000, E1  +428.240, E3 -178840.056}
SPL {X  -159.990, Y  +610.177, Z    +0.000, E1  +428.265, E3 -178852.043}
SPL {X  -159.990, Y  +627.954, Z    +0.000, E1  +428.256, E3 -178867.114}
SPL {X  -159.990, Y  +644.561, Z    +0.000, E1  +428.258, E3 -178881.166}
SPL {X  -159.990, Y  +661.441, Z    +0.000, E1  +428.256, E3 -178895.475}
SPL {X  -159.958, Y  +674.683, Z    +0.000, E1  +428.238, E3 -178906.738}
SPL {X  -159.269, Y  +686.675, Z    +0.000, E1  +428.163, E3 -178917.615}
SPL {X  -158.119, Y  +695.895, Z    +0.000, E1  +428.003, E3 -178926.656}
SPL {X  -156.550, Y  +704.498, Z    +0.000, E1  +427.821, E3 -178935.546}
SPL {X  -153.468, Y  +716.715, Z    +0.000, E1  +427.444, E3 -178949.009}
SPL {X  -149.840, Y  +727.578, Z    +0.000, E1  +426.935, E3 -178961.885}
SPL {X  -145.768, Y  +737.444, Z    +0.000, E1  +426.379, E3 -178974.187}
SPL {X  -141.751, Y  +745.686, Z    +0.000, E1  +425.756, E3 -178985.003}
SPL {X  -138.928, Y  +750.847, Z    +0.000, E1  +425.305, E3 -178991.973}
SPL {X  -135.390, Y  +756.743, Z    +0.000, E1  +424.775, E3 -179000.005}
SPL {X  -132.002, Y  +761.900, Z    +0.000, E1  +424.179, E3 -179007.236}
SPL {X  -128.512, Y  +766.796, Z    +0.000, E1  +423.597, E3 -179014.091}
SPL {X   -99.023, Y  +797.163, Z    +0.000, E1  +413.965, E3 -179115.920}
ENDSPLINE

SPLINE
SPL {X  -130.021, Y  +764.727, Z    +0.000, E1  +405.990, E3 -179255.440}
SPL {X  -148.409, Y  +731.264, Z    +0.000, E1  +396.685, E3 -179279.153}
SPL {X  -155.017, Y  +711.078, Z    +0.000, E1  +387.846, E3 -179286.214}
SPL {X  -158.217, Y  +695.254, Z    +0.000, E1  +378.896, E3 -179289.657}
SPL {X  -159.524, Y  +683.703, Z    +0.000, E1  +371.166, E3 -179291.099}
SPL {X  -159.986, Y  +672.621, Z    +0.000, E1  +362.847, E3 -179291.741}
SPL {X  -159.990, Y  +669.426, Z    +0.000, E1  +359.932, E3 -179291.799}
SPL {X  -159.990, Y  +666.879, Z    +0.000, E1  +356.292, E3 -179291.847}
SPL {X  -159.990, Y  +662.620, Z    +0.000, E1  +348.758, E3 -179292.048}
SPL {X  -159.990, Y  +657.714, Z    +0.000, E1  +339.502, E3 -179292.469}
SPL {X  -159.990, Y  +651.038, Z    +0.000, E1  +327.797, E3 -179293.372}
SPL {X  -159.990, Y  +637.243, Z    +0.000, E1  +311.500, E3 -179296.497}
SPL {X  -159.990, Y  +579.875, Z    +0.000, E1  +294.421, E3 -179319.356}
SPL {X  -159.990, Y  +453.091, Z    +0.000, E1  +291.862, E3 -179402.325}
SPL {X  -159.990, Y  +434.933, Z    +0.000, E1  +291.864, E3 -179417.819}
SPL {X  -159.990, Y  +420.071, Z    +0.000, E1  +291.886, E3 -179430.545}
SPL {X  -159.990, Y  +408.047, Z    +0.000, E1  +291.885, E3 -179440.792}
SPL {X  -159.990, Y  +395.904, Z    +0.000, E1  +291.881, E3 -179451.128}
SPL {X  -158.518, Y  +360.846, Z    +0.000, E1  +289.610, E3 -179459.064}
SPL {X  -157.390, Y  +353.775, Z    +0.000, E1  +289.868, E3 -179466.740}
SPL {X  -156.475, Y  +349.148, Z    +0.000, E1  +290.612, E3 -179476.902}
SPL {X  -155.786, Y  +346.063, Z    +0.000, E1  +291.892, E3 -179490.196}
SPL {X  -154.401, Y  +340.583, Z    +0.000, E1  +292.675, E3 -179500.893}
SPL {X  -152.032, Y  +332.668, Z    +0.000, E1  +292.988, E3 -179510.069}
SPL {X  -148.460, Y  +322.864, Z    +0.000, E1  +293.452, E3 -179521.951}
SPL {X  -144.472, Y  +313.764, Z    +0.000, E1  +294.050, E3 -179533.615}
SPL {X  -141.765, Y  +308.342, Z    +0.000, E1  +294.475, E3 -179540.812}
SPL {X  -139.838, Y  +304.768, Z    +0.000, E1  +294.773, E3 -179545.631}
SPL {X  -137.162, Y  +300.138, Z    +0.000, E1  +295.180, E3 -179551.937}
SPL {X  -132.996, Y  +293.568, Z    +0.000, E1  +295.842, E3 -179561.072}
SPL {X  -128.628, Y  +287.360, Z    +0.000, E1  +296.617, E3 -179569.873}
SPL {X   -98.696, Y  +256.580, Z    +0.000, E1  +308.006, E3 -179706.991}
ENDSPLINE

SPLINE
SPL {X  -138.661, Y  +302.689, Z    +0.000, E1  +316.811, E3 -179824.720}
SPL {X  -154.202, Y  +339.857, Z    +0.000, E1  +330.366, E3 -179842.373}
SPL {X  -158.556, Y  +361.128, Z    +0.000, E1  +342.470, E3 -179846.894}
SPL {X  -159.866, Y  +376.206, Z    +0.000, E1  +353.031, E3 -179848.423}
SPL {X  -159.990, Y  +384.326, Z    +0.000, E1  +359.760, E3 -179848.696}
SPL {X  -159.990, Y  +385.649, Z    +0.000, E1  +361.559, E3 -179848.709}
SPL {X  -159.990, Y  +388.306, Z    +0.000, E1  +365.901, E3 -179848.780}
SPL {X  -159.990, Y  +392.624, Z    +0.000, E1  +373.655, E3 -179849.029}
SPL {X  -159.990, Y  +398.511, Z    +0.000, E1  +384.979, E3 -179849.610}
SPL {X  -159.990, Y  +405.629, Z    +0.000, E1  +396.596, E3 -179850.740}
SPL {X  -159.990, Y  +418.631, Z    +0.000, E1  +410.627, E3 -179853.688}
SPL {X  -159.990, Y  +468.459, Z    +0.000, E1  +425.348, E3 -179873.231}
SPL {X  -159.990, Y  +601.948, Z    +0.000, E1  +428.261, E3 -179959.357}
SPL {X  -159.990, Y  +619.726, Z    +0.000, E1  +428.262, E3 -179974.418}
SPL {X  -159.990, Y  +636.530, Z    +0.000, E1  +428.257, E3 -179988.654}
SPL {X  -159.990, Y  +653.116, Z    +0.000, E1  +428.255, E3 -180002.710}
SPL {X  -159.990, Y  +670.874, Z    +0.000, E1  +428.264, E3 -180017.725}
SPL {X  -159.269, Y  +686.675, Z    +0.000, E1  +428.163, E3 -180031.901}
SPL {X  -157.606, Y  +699.018, Z    +0.000, E1  +427.957, E3 -180044.085}
SPL {X  -155.210, Y  +710.317, Z    +0.000, E1  +427.656, E3 -180056.125}
SPL {X  -152.048, Y  +721.282, Z    +0.000, E1  +427.243, E3 -180068.617}
SPL {X  -148.485, Y  +731.073, Z    +0.000, E1  +426.748, E3 -180080.466}
SPL {X  -145.075, Y  +738.953, Z    +0.000, E1  +426.252, E3 -180090.458}
SPL {X  -141.751, Y  +745.686, Z    +0.000, E1  +425.756, E3 -180099.289}
SPL {X  -138.928, Y  +750.847, Z    +0.000, E1  +425.305, E3 -180106.258}
SPL {X  -136.328, Y  +755.234, Z    +0.000, E1  +424.898, E3 -180112.249}
SPL {X  -132.717, Y  +760.848, Z    +0.000, E1  +424.322, E3 -180120.022}
SPL {X  -128.512, Y  +766.796, Z    +0.000, E1  +423.597, E3 -180128.376}
SPL {X   -99.023, Y  +797.163, Z    +0.000, E1  +413.965, E3 -180230.206}
ENDSPLINE

SPLINE
SPL {X  -130.021, Y  +764.727, Z    +0.000, E1  +405.990, E3 -180369.725}
SPL {X  -148.409, Y  +731.264, Z    +0.000, E1  +396.685, E3 -180393.439}
SPL {X  -155.017, Y  +711.078, Z    +0.000, E1  +387.846, E3 -180400.500}
SPL {X  -158.217, Y  +695.254, Z    +0.000, E1  +378.896, E3 -180403.943}
SPL {X  -159.762, Y  +680.037, Z    +0.000, E1  +368.585, E3 -180405.660}
SPL {X  -159.990, Y  +671.255, Z    +0.000, E1  +361.602, E3 -180406.065}
SPL {X  -159.990, Y  +669.426, Z    +0.000, E1  +359.932, E3 -180406.085}
SPL {X  -159.990, Y  +666.879, Z    +0.000, E1  +356.292, E3 -180406.133}
SPL {X  -159.990, Y  +662.620, Z    +0.000, E1  +348.758, E3 -180406.334}
SPL {X  -159.990, Y  +657.714, Z    +0.000, E1  +339.502, E3 -180406.755}
SPL {X  -159.990, Y  +651.038, Z    +0.000, E1  +327.797, E3 -180407.658}
SPL {X  -159.990, Y  +637.243, Z    +0.000, E1  +311.500, E3 -180410.783}
SPL {X  -159.990, Y  +579.875, Z    +0.000, E1  +294.421, E3 -180433.641}
SPL {X  -159.990, Y  +453.091, Z    +0.000, E1  +291.862, E3 -180516.611}
SPL {X  -159.990, Y  +434.933, Z    +0.000, E1  +291.864, E3 -180532.105}
SPL {X  -159.990, Y  +420.071, Z    +0.000, E1  +291.886, E3 -180544.831}
SPL {X  -159.990, Y  +408.047, Z    +0.000, E1  +291.885, E3 -180555.078}
SPL {X  -159.990, Y  +395.904, Z    +0.000, E1  +291.881, E3 -180565.414}
SPL {X  -157.896, Y  +356.699, Z    +0.000, E1  +289.725, E3 -180577.724}
SPL {X  -156.475, Y  +349.148, Z    +0.000, E1  +290.612, E3 -180591.188}
SPL {X  -155.960, Y  +346.816, Z    +0.000, E1  +291.495, E3 -180600.349}
SPL {X  -154.913, Y  +342.515, Z    +0.000, E1  +292.501, E3 -180612.363}
SPL {X  -152.032, Y  +332.668, Z    +0.000, E1  +292.988, E3 -180624.354}
SPL {X  -148.460, Y  +322.864, Z    +0.000, E1  +293.452, E3 -180636.237}
SPL {X  -144.472, Y  +313.764, Z    +0.000, E1  +294.050, E3 -180647.900}
SPL {X  -140.755, Y  +306.442, Z    +0.000, E1  +294.606, E3 -180657.615}
SPL {X  -137.162, Y  +300.138, Z    +0.000, E1  +295.180, E3 -180666.223}
SPL {X  -134.303, Y  +295.555, Z    +0.000, E1  +295.659, E3 -180672.604}
SPL {X  -131.069, Y  +290.753, Z    +0.000, E1  +296.178, E3 -180679.338}
SPL {X  -127.815, Y  +286.271, Z    +0.000, E1  +296.784, E3 -180685.726}
SPL {X   -98.696, Y  +256.580, Z    +0.000, E1  +308.006, E3 -180821.277}
ENDSPLINE

SPLINE
SPL {X  -138.661, Y  +302.689, Z    +0.000, E1  +316.811, E3 -180939.005}
SPL {X  -154.202, Y  +339.857, Z    +0.000, E1  +330.366, E3 -180956.658}
SPL {X  -158.556, Y  +361.128, Z    +0.000, E1  +342.470, E3 -180961.180}
SPL {X  -159.663, Y  +372.278, Z    +0.000, E1  +350.186, E3 -180962.461}
SPL {X  -159.986, Y  +381.388, Z    +0.000, E1  +357.201, E3 -180962.933}
SPL {X  -159.990, Y  +384.492, Z    +0.000, E1  +359.986, E3 -180962.983}
SPL {X  -159.990, Y  +385.649, Z    +0.000, E1  +361.559, E3 -180962.994}
SPL {X  -159.990, Y  +389.563, Z    +0.000, E1  +367.931, E3 -180963.127}
SPL {X  -159.990, Y  +396.421, Z    +0.000, E1  +380.831, E3 -180963.672}
SPL {X  -159.990, Y  +405.629, Z    +0.000, E1  +396.596, E3 -180965.026}
SPL {X  -159.990, Y  +418.631, Z    +0.000, E1  +410.627, E3 -180967.973}
SPL {X  -159.990, Y  +468.459, Z    +0.000, E1  +425.348, E3 -180987.517}
SPL {X  -159.990, Y  +601.948, Z    +0.000, E1  +428.261, E3 -181073.643}
SPL {X  -159.990, Y  +619.726, Z    +0.000, E1  +428.262, E3 -181088.704}
SPL {X  -159.990, Y  +636.530, Z    +0.000, E1  +428.257, E3 -181102.940}
SPL {X  -159.990, Y  +648.825, Z    +0.000, E1  +428.237, E3 -181113.398}
SPL {X  -159.990, Y  +661.441, Z    +0.000, E1  +428.256, E3 -181124.047}
SPL {X  -159.958, Y  +674.683, Z    +0.000, E1  +428.238, E3 -181135.309}
SPL {X  -159.269, Y  +686.675, Z    +0.000, E1  +428.163, E3 -181146.187}
SPL {X  -157.606, Y  +699.018, Z    +0.000, E1  +427.957, E3 -181158.370}
SPL {X  -155.210, Y  +710.317, Z    +0.000, E1  +427.656, E3 -181170.410}
SPL {X  -152.048, Y  +721.282, Z    +0.000, E1  +427.243, E3 -181182.903}
SPL {X  -148.485, Y  +731.073, Z    +0.000, E1  +426.748, E3 -181194.752}
SPL {X  -145.075, Y  +738.953, Z    +0.000, E1  +426.252, E3 -181204.744}
SPL {X  -141.751, Y  +745.686, Z    +0.000, E1  +425.756, E3 -181213.575}
SPL {X  -138.928, Y  +750.847, Z    +0.000, E1  +425.305, E3 -181220.544}
SPL {X  -136.328, Y  +755.234, Z    +0.000, E1  +424.898, E3 -181226.534}
SPL {X  -132.717, Y  +760.848, Z    +0.000, E1  +424.322, E3 -181234.308}
SPL {X  -128.512, Y  +766.796, Z    +0.000, E1  +423.597, E3 -181242.662}
SPL {X   -99.023, Y  +797.163, Z    +0.000, E1  +413.965, E3 -181344.492}
ENDSPLINE

SPLINE
SPL {X  -130.021, Y  +764.727, Z    +0.000, E1  +405.990, E3 -181484.011}
SPL {X  -148.409, Y  +731.264, Z    +0.000, E1  +396.685, E3 -181507.725}
SPL {X  -155.017, Y  +711.078, Z    +0.000, E1  +387.846, E3 -181514.786}
SPL {X  -158.217, Y  +695.254, Z    +0.000, E1  +378.896, E3 -181518.228}
SPL {X  -159.762, Y  +680.037, Z    +0.000, E1  +368.585, E3 -181519.945}
SPL {X  -159.990, Y  +671.255, Z    +0.000, E1  +361.602, E3 -181520.351}
SPL {X  -159.990, Y  +669.426, Z    +0.000, E1  +359.932, E3 -181520.371}
SPL {X  -159.990, Y  +666.879, Z    +0.000, E1  +356.292, E3 -181520.418}
SPL {X  -159.990, Y  +662.620, Z    +0.000, E1  +348.758, E3 -181520.620}
SPL {X  -159.990, Y  +657.714, Z    +0.000, E1  +339.502, E3 -181521.041}
SPL {X  -159.990, Y  +651.038, Z    +0.000, E1  +327.797, E3 -181521.943}
SPL {X  -159.990, Y  +637.243, Z    +0.000, E1  +311.500, E3 -181525.068}
SPL {X  -159.990, Y  +579.875, Z    +0.000, E1  +294.421, E3 -181547.927}
SPL {X  -159.990, Y  +453.091, Z    +0.000, E1  +291.862, E3 -181630.897}
SPL {X  -159.990, Y  +434.933, Z    +0.000, E1  +291.864, E3 -181646.390}
SPL {X  -159.990, Y  +420.071, Z    +0.000, E1  +291.886, E3 -181659.116}
SPL {X  -159.990, Y  +408.047, Z    +0.000, E1  +291.885, E3 -181669.364}
SPL {X  -159.990, Y  +395.904, Z    +0.000, E1  +291.881, E3 -181679.700}
SPL {X  -157.896, Y  +356.699, Z    +0.000, E1  +289.725, E3 -181692.009}
SPL {X  -156.475, Y  +349.148, Z    +0.000, E1  +290.612, E3 -181705.473}
SPL {X  -155.756, Y  +345.937, Z    +0.000, E1  +291.895, E3 -181718.904}
ENDSPLINE

SPLINE
SPL {X  -159.342, Y  +368.120, Z    +0.000, E1  +296.535, E3 -181733.283}
ENDSPLINE

SPLINE
SPL {X  -158.431, Y  +360.219, Z    +0.000, E1  +296.670, E3 -181742.607}
SPL {X  -156.653, Y  +349.995, Z    +0.000, E1  +296.892, E3 -181755.176}
SPL {X  -153.792, Y  +338.401, Z    +0.000, E1  +297.323, E3 -181770.345}
SPL {X  -151.244, Y  +330.327, Z    +0.000, E1  +297.748, E3 -181781.498}
SPL {X  -148.909, Y  +323.994, Z    +0.000, E1  +298.107, E3 -181790.484}
SPL {X  -146.667, Y  +318.581, Z    +0.000, E1  +298.485, E3 -181798.404}
SPL {X  -144.416, Y  +313.647, Z    +0.000, E1  +298.845, E3 -181805.740}
SPL {X  -141.484, Y  +307.808, Z    +0.000, E1  +299.342, E3 -181814.633}
SPL {X  -139.055, Y  +303.377, Z    +0.000, E1  +299.788, E3 -181821.546}
SPL {X  -136.464, Y  +298.988, Z    +0.000, E1  +300.231, E3 -181828.420}
SPL {X  -133.486, Y  +294.305, Z    +0.000, E1  +300.785, E3 -181835.882}
SPL {X  -111.198, Y  +267.470, Z    +0.000, E1  +308.990, E3 -181936.902}
ENDSPLINE

SPLINE
SPL {X  -136.508, Y  +299.059, Z    +0.000, E1  +318.212, E3 -182047.839}
SPL {X  -153.176, Y  +336.305, Z    +0.000, E1  +330.872, E3 -182074.404}
SPL {X  -158.263, Y  +359.056, Z    +0.000, E1  +342.551, E3 -182081.078}
SPL {X  -159.616, Y  +371.564, Z    +0.000, E1  +350.434, E3 -182082.983}
SPL {X  -159.983, Y  +381.031, Z    +0.000, E1  +357.053, E3 -182083.674}
SPL {X  -159.990, Y  +384.524, Z    +0.000, E1  +359.995, E3 -182083.762}
SPL {X  -159.990, Y  +386.890, Z    +0.000, E1  +362.742, E3 -182083.818}
SPL {X  -159.990, Y  +392.248, Z    +0.000, E1  +370.895, E3 -182084.145}
SPL {X  -159.990, Y  +398.030, Z    +0.000, E1  +380.706, E3 -182084.797}
SPL {X  -159.990, Y  +404.858, Z    +0.000, E1  +391.125, E3 -182086.041}
SPL {X  -159.990, Y  +416.328, Z    +0.000, E1  +404.105, E3 -182088.978}
SPL {X  -159.990, Y  +459.824, Z    +0.000, E1  +420.326, E3 -182108.900}
SPL {X  -159.990, Y  +565.974, Z    +0.000, E1  +423.959, E3 -182192.389}
SPL {X  -159.990, Y  +578.588, Z    +0.000, E1  +423.918, E3 -182205.568}
SPL {X  -159.990, Y  +590.041, Z    +0.000, E1  +423.939, E3 -182217.423}
SPL {X  -159.990, Y  +601.352, Z    +0.000, E1  +423.918, E3 -182229.209}
SPL {X  -159.990, Y  +610.973, Z    +0.000, E1  +423.927, E3 -182239.177}
SPL {X  -159.990, Y  +624.756, Z    +0.000, E1  +423.949, E3 -182253.455}
SPL {X  -159.990, Y  +640.674, Z    +0.000, E1  +423.943, E3 -182269.992}
SPL {X  -159.990, Y  +652.355, Z    +0.000, E1  +423.915, E3 -182282.191}
SPL {X  -159.990, Y  +665.748, Z    +0.000, E1  +423.953, E3 -182296.044}
SPL {X  -159.643, Y  +682.032, Z    +0.000, E1  +423.894, E3 -182313.337}
SPL {X  -158.070, Y  +696.212, Z    +0.000, E1  +423.682, E3 -182329.676}
SPL {X  -155.481, Y  +709.215, Z    +0.000, E1  +423.310, E3 -182345.867}
SPL {X  -153.138, Y  +717.820, Z    +0.000, E1  +422.909, E3 -182357.285}
SPL {X  -151.229, Y  +723.716, Z    +0.000, E1  +422.630, E3 -182365.295}
SPL {X  -148.422, Y  +731.231, Z    +0.000, E1  +422.207, E3 -182375.853}
SPL {X  -145.802, Y  +737.367, Z    +0.000, E1  +421.758, E3 -182384.806}
SPL {X  -143.476, Y  +742.291, Z    +0.000, E1  +421.379, E3 -182392.106}
SPL {X  -141.015, Y  +747.074, Z    +0.000, E1  +420.958, E3 -182399.363}
SPL {X  -138.539, Y  +751.523, Z    +0.000, E1  +420.526, E3 -182406.197}
SPL {X  -136.299, Y  +755.281, Z    +0.000, E1  +420.128, E3 -182412.059}
SPL {X  -133.306, Y  +759.967, Z    +0.000, E1  +419.584, E3 -182419.453}
SPL {X  -112.019, Y  +785.730, Z    +0.000, E1  +410.795, E3 -182522.194}
ENDSPLINE

SPLINE
SPL {X  -138.335, Y  +751.876, Z    +0.000, E1  +401.001, E3 -182636.492}
SPL {X  -150.285, Y  +726.376, Z    +0.000, E1  +392.667, E3 -182654.901}
SPL {X  -154.601, Y  +712.673, Z    +0.000, E1  +386.751, E3 -182660.506}
SPL {X  -158.303, Y  +694.673, Z    +0.000, E1  +377.238, E3 -182665.175}
SPL {X  -159.774, Y  +679.819, Z    +0.000, E1  +367.840, E3 -182667.250}
SPL {X  -159.990, Y  +671.106, Z    +0.000, E1  +361.459, E3 -182667.770}
SPL {X  -159.990, Y  +669.154, Z    +0.000, E1  +359.694, E3 -182667.802}
SPL {X  -159.990, Y  +666.004, Z    +0.000, E1  +355.742, E3 -182667.902}
SPL {X  -159.990, Y  +661.286, Z    +0.000, E1  +348.294, E3 -182668.218}
SPL {X  -159.990, Y  +656.470, Z    +0.000, E1  +340.220, E3 -182668.756}
SPL {X  -159.990, Y  +651.555, Z    +0.000, E1  +332.416, E3 -182669.563}
SPL {X  -159.990, Y  +640.109, Z    +0.000, E1  +318.471, E3 -182672.392}
SPL {X  -159.990, Y  +589.014, Z    +0.000, E1  +298.500, E3 -182694.258}
SPL {X  -159.990, Y  +484.717, Z    +0.000, E1  +295.169, E3 -182772.441}
SPL {X  -159.990, Y  +474.300, Z    +0.000, E1  +295.184, E3 -182782.869}
SPL {X  -159.990, Y  +460.248, Z    +0.000, E1  +295.138, E3 -182796.779}
SPL {X  -159.990, Y  +443.816, Z    +0.000, E1  +295.158, E3 -182813.194}
SPL {X  -159.990, Y  +410.689, Z    +0.000, E1  +292.263, E3 -182820.918}
SPL {X  -159.990, Y  +399.563, Z    +0.000, E1  +292.427, E3 -182832.157}
SPL {X  -159.990, Y  +393.786, Z    +0.000, E1  +293.391, E3 -182845.146}
SPL {X  -159.990, Y  +387.038, Z    +0.000, E1  +293.844, E3 -182855.002}
SPL {X  -159.983, Y  +380.995, Z    +0.000, E1  +294.559, E3 -182866.570}
SPL {X  -159.898, Y  +377.064, Z    +0.000, E1  +295.481, E3 -182877.384}
SPL {X  -159.533, Y  +370.414, Z    +0.000, E1  +296.253, E3 -182890.381}
SPL {X  -158.431, Y  +360.219, Z    +0.000, E1  +296.670, E3 -182903.898}
SPL {X  -157.299, Y  +353.279, Z    +0.000, E1  +296.835, E3 -182912.394}
SPL {X  -155.242, Y  +343.812, Z    +0.000, E1  +297.102, E3 -182924.442}
SPL {X  -151.999, Y  +332.569, Z    +0.000, E1  +297.592, E3 -182939.601}
SPL {X  -148.909, Y  +323.994, Z    +0.000, E1  +298.107, E3 -182951.774}
SPL {X  -146.667, Y  +318.581, Z    +0.000, E1  +298.485, E3 -182959.694}
SPL {X  -144.416, Y  +313.647, Z    +0.000, E1  +298.845, E3 -182967.031}
SPL {X  -141.484, Y  +307.808, Z    +0.000, E1  +299.342, E3 -182975.924}
SPL {X  -139.055, Y  +303.377, Z    +0.000, E1  +299.788, E3 -182982.836}
SPL {X  -136.464, Y  +298.988, Z    +0.000, E1  +300.231, E3 -182989.710}
SPL {X  -133.486, Y  +294.305, Z    +0.000, E1  +300.785, E3 -182997.172}
SPL {X  -111.198, Y  +267.470, Z    +0.000, E1  +308.990, E3 -183098.193}
ENDSPLINE

